LIN {X 0,Y 474.615,Z 281.367,A -85,B 0,C 180,E1 -7440.886,E2 -7440.886} C_VEL
LIN {X 0,Y 474.653,Z 281.359,A -85,B 0,C 180,E1 -7443.629,E2 -7443.629} C_VEL
LIN {X 0,Y 474.629,Z 281.364,A -85,B 0,C 180,E1 -7446.642,E2 -7446.642} C_VEL
LIN {X 0,Y 474.65,Z 281.358,A -85,B 0,C 180,E1 -7450.09,E2 -7450.09} C_VEL
LIN {X 0,Y 474.651,Z 281.358,A -85,B 0,C 180,E1 -7451.7,E2 -7451.7} C_VEL
LIN {X 0,Y 473.99,Z 281.443,A -85,B 0,C 180,E1 -7452.409,E2 -7452.409} C_VEL
LIN {X 0,Y 471.138,Z 281.798,A -85,B 0,C 180,E1 -7453.561,E2 -7453.561} C_VEL
LIN {X 0,Y 468.72,Z 282.101,A -85,B 0,C 180,E1 -7454.489,E2 -7454.489} C_VEL
LIN {X 0,Y 467.679,Z 282.229,A -85,B 0,C 180,E1 -7455.206,E2 -7455.206} C_VEL
LIN {X 0,Y 467.593,Z 282.238,A -85,B 0,C 180,E1 -7455.449,E2 -7455.449} C_VEL
LIN {X 0,Y 467.65,Z 282.234,A -85,B 0,C 180,E1 -7458.734,E2 -7458.734} C_VEL
LIN {X 0,Y 467.747,Z 282.218,A -85,B 0,C 180,E1 -7462.228,E2 -7462.228} C_VEL
LIN {X 0,Y 467.722,Z 282.226,A -85,B 0,C 180,E1 -7464.827,E2 -7464.827} C_VEL
LIN {X 0,Y 467.857,Z 282.206,A -85,B 0,C 180,E1 -7467.416,E2 -7467.416} C_VEL
LIN {X 0,Y 467.88,Z 282.201,A -85,B 0,C 180,E1 -7469.999,E2 -7469.999} C_VEL
LIN {X 0,Y 467.857,Z 282.206,A -85,B 0,C 180,E1 -7472.581,E2 -7472.581} C_VEL
LIN {X 0,Y 467.731,Z 282.219,A -85,B 0,C 180,E1 -7476.036,E2 -7476.036} C_VEL
LIN {X 0,Y 467.676,Z 282.228,A -85,B 0,C 180,E1 -7478.641,E2 -7478.641} C_VEL
LIN {X 0,Y 467.675,Z 282.226,A -85,B 0,C 180,E1 -7482.142,E2 -7482.142} C_VEL
LIN {X 0,Y 467.64,Z 282.231,A -85,B 0,C 180,E1 -7485.883,E2 -7485.883} C_VEL
LIN {X 0,Y 467.613,Z 282.238,A -85,B 0,C 180,E1 -7489.305,E2 -7489.305} C_VEL
LIN {X 0,Y 467.553,Z 282.241,A -85,B 0,C 180,E1 -7492.069,E2 -7492.069} C_VEL
LIN {X 0,Y 467.59,Z 282.241,A -85,B 0,C 180,E1 -7494.884,E2 -7494.884} C_VEL
LIN {X 0,Y 467.61,Z 282.235,A -85,B 0,C 180,E1 -7497.765,E2 -7497.765} C_VEL
LIN {X 0,Y 467.558,Z 282.246,A -85,B 0,C 180,E1 -7501.044,E2 -7501.044} C_VEL
LIN {X 0,Y 467.566,Z 282.239,A -85,B 0,C 180,E1 -7504.239,E2 -7504.239} C_VEL
LIN {X 0,Y 467.526,Z 282.252,A -85,B 0,C 180,E1 -7507.184,E2 -7507.184} C_VEL
LIN {X 0,Y 467.572,Z 282.24,A -85,B 0,C 180,E1 -7510.258,E2 -7510.258} C_VEL
LIN {X 0,Y 467.639,Z 282.299,A -85,B 0,C 180,E1 -7512.891,E2 -7512.891} C_VEL
LIN {X 0,Y 468.46,Z 287.03,A -85,B 0,C 180,E1 -7513.937,E2 -7513.937} C_VEL
LIN {X 0,Y 468.452,Z 292.664,A -85,B 0,C 180,E1 -7515.1,E2 -7515.1} C_VEL
LIN {X 0,Y 471.354,Z 307.156,A -85,B 0,C 180,E1 -7515.447,E2 -7515.447} C_VEL
LIN {X 0,Y 470.368,Z 400.533,A -85,B 0,C 180,E1 -7516.983,E2 -7516.983} C_VEL
LIN {X 0,Y 470.151,Z 413.603,A -85,B 0,C 180,E1 -7517.376,E2 -7517.376} C_VEL
LIN {X 0,Y 469.792,Z 425.843,A -85,B 0,C 180,E1 -7517.909,E2 -7517.909} C_VEL
LIN {X 0,Y 469.379,Z 437.833,A -85,B 0,C 180,E1 -7518.619,E2 -7518.619} C_VEL
LIN {X 0,Y 468.918,Z 448.857,A -85,B 0,C 180,E1 -7519.452,E2 -7519.452} C_VEL
LIN {X 0,Y 468.501,Z 458.862,A -85,B 0,C 180,E1 -7520.392,E2 -7520.392} C_VEL
LIN {X 0,Y 468.086,Z 468.527,A -85,B 0,C 180,E1 -7521.514,E2 -7521.514} C_VEL
LIN {X 0,Y 467.678,Z 477.339,A -85,B 0,C 180,E1 -7522.783,E2 -7522.783} C_VEL
LIN {X 0,Y 467.324,Z 484.669,A -85,B 0,C 180,E1 -7524.091,E2 -7524.091} C_VEL
LIN {X 0,Y 467.094,Z 490.987,A -85,B 0,C 180,E1 -7525.526,E2 -7525.526} C_VEL
LIN {X 0,Y 466.941,Z 495.005,A -85,B 0,C 180,E1 -7526.677,E2 -7526.677} C_VEL
LIN {X 0,Y 466.833,Z 498.969,A -85,B 0,C 180,E1 -7528.204,E2 -7528.204} C_VEL
LIN {X 0,Y 466.675,Z 500.847,A -85,B 0,C 180,E1 -7529.201,E2 -7529.201} C_VEL
LIN {X 0,Y 466.619,Z 502.698,A -85,B 0,C 180,E1 -7530.863,E2 -7530.863} C_VEL
LIN {X 0,Y 466.607,Z 503.037,A -85,B 0,C 180,E1 -7532.69,E2 -7532.69} C_VEL
LIN {X 0,Y 466.652,Z 502.053,A -85,B 0,C 180,E1 -7534.104,E2 -7534.104} C_VEL
LIN {X 0,Y 466.727,Z 500.735,A -85,B 0,C 180,E1 -7535.063,E2 -7535.063} C_VEL
LIN {X 0,Y 466.906,Z 497.465,A -85,B 0,C 180,E1 -7536.646,E2 -7536.646} C_VEL
LIN {X 0,Y 467.021,Z 493.781,A -85,B 0,C 180,E1 -7537.901,E2 -7537.901} C_VEL
LIN {X 0,Y 467.222,Z 488.421,A -85,B 0,C 180,E1 -7539.306,E2 -7539.306} C_VEL
LIN {X 0,Y 467.566,Z 481.593,A -85,B 0,C 180,E1 -7540.69,E2 -7540.69} C_VEL
LIN {X 0,Y 467.971,Z 473.014,A -85,B 0,C 180,E1 -7542.07,E2 -7542.07} C_VEL
LIN {X 0,Y 468.422,Z 464.162,A -85,B 0,C 180,E1 -7543.213,E2 -7543.213} C_VEL
LIN {X 0,Y 468.804,Z 454.996,A -85,B 0,C 180,E1 -7544.18,E2 -7544.18} C_VEL
LIN {X 0,Y 469.327,Z 443.665,A -85,B 0,C 180,E1 -7545.141,E2 -7545.141} C_VEL
LIN {X 0,Y 469.742,Z 431.9,A -85,B 0,C 180,E1 -7545.93,E2 -7545.93} C_VEL
LIN {X 0,Y 470.084,Z 419.99,A -85,B 0,C 180,E1 -7546.532,E2 -7546.532} C_VEL
LIN {X 0,Y 470.378,Z 407.324,A -85,B 0,C 180,E1 -7546.992,E2 -7546.992} C_VEL
LIN {X 0,Y 470.57,Z 395.176,A -85,B 0,C 180,E1 -7547.274,E2 -7547.274} C_VEL
LIN {X 0,Y 471.399,Z 305.966,A -85,B 0,C 180,E1 -7548.757,E2 -7548.757} C_VEL
LIN {X 0,Y 468.554,Z 292.044,A -85,B 0,C 180,E1 -7549.139,E2 -7549.139} C_VEL
LIN {X 0,Y 468.454,Z 286.338,A -85,B 0,C 180,E1 -7550.066,E2 -7550.066} C_VEL
LIN {X 0,Y 467.639,Z 282.237,A -85,B 0,C 180,E1 -7550.785,E2 -7550.785} C_VEL
LIN {X 0,Y 467.643,Z 282.237,A -85,B 0,C 180,E1 -7553.095,E2 -7553.095} C_VEL
LIN {X 0,Y 467.666,Z 282.236,A -85,B 0,C 180,E1 -7554.827,E2 -7554.827} C_VEL
LIN {X 0,Y 467.807,Z 282.215,A -85,B 0,C 180,E1 -7557.417,E2 -7557.417} C_VEL
LIN {X 0,Y 467.77,Z 282.221,A -85,B 0,C 180,E1 -7560.861,E2 -7560.861} C_VEL
LIN {X 0,Y 467.808,Z 282.214,A -85,B 0,C 180,E1 -7562.584,E2 -7562.584} C_VEL
LIN {X 0,Y 467.688,Z 282.225,A -85,B 0,C 180,E1 -7566.039,E2 -7566.039} C_VEL
LIN {X 0,Y 467.627,Z 282.235,A -85,B 0,C 180,E1 -7568.644,E2 -7568.644} C_VEL
LIN {X 0,Y 467.643,Z 282.23,A -85,B 0,C 180,E1 -7572.146,E2 -7572.146} C_VEL
LIN {X 0,Y 467.597,Z 282.235,A -85,B 0,C 180,E1 -7575.888,E2 -7575.888} C_VEL
LIN {X 0,Y 467.571,Z 282.241,A -85,B 0,C 180,E1 -7579.31,E2 -7579.31} C_VEL
LIN {X 0,Y 467.483,Z 282.249,A -85,B 0,C 180,E1 -7582.077,E2 -7582.077} C_VEL
LIN {X 0,Y 467.555,Z 282.246,A -85,B 0,C 180,E1 -7584.89,E2 -7584.89} C_VEL
LIN {X 0,Y 467.582,Z 282.238,A -85,B 0,C 180,E1 -7587.772,E2 -7587.772} C_VEL
LIN {X 0,Y 467.524,Z 282.25,A -85,B 0,C 180,E1 -7591.048,E2 -7591.048} C_VEL
LIN {X 0,Y 467.549,Z 282.239,A -85,B 0,C 180,E1 -7594.246,E2 -7594.246} C_VEL
LIN {X 0,Y 467.511,Z 282.25,A -85,B 0,C 180,E1 -7597.19,E2 -7597.19} C_VEL
LIN {X 0,Y 467.563,Z 282.239,A -85,B 0,C 180,E1 -7600.267,E2 -7600.267} C_VEL
LIN {X 0,Y 467.555,Z 282.239,A -85,B 0,C 180,E1 -7602.571,E2 -7602.571} C_VEL
LIN {X 0,Y 467.54,Z 282.246,A -85,B 0,C 180,E1 -7605.057,E2 -7605.057} C_VEL
LIN {X 0,Y 467.562,Z 282.246,A -85,B 0,C 180,E1 -7607.444,E2 -7607.444} C_VEL
LIN {X 0,Y 467.535,Z 282.246,A -85,B 0,C 180,E1 -7610.857,E2 -7610.857} C_VEL
LIN {X 0,Y 467.539,Z 282.246,A -85,B 0,C 180,E1 -7614.265,E2 -7614.265} C_VEL
LIN {X 0,Y 467.563,Z 282.251,A -85,B 0,C 180,E1 -7617.325,E2 -7617.325} C_VEL
LIN {X 0,Y 467.543,Z 282.248,A -85,B 0,C 180,E1 -7620.674,E2 -7620.674} C_VEL
LIN {X 0,Y 467.63,Z 282.33,A -85,B 0,C 180,E1 -7623.686,E2 -7623.686} C_VEL
LIN {X 0,Y 469.549,Z 292.668,A -85,B 0,C 180,E1 -7625.432,E2 -7625.432} C_VEL
LIN {X 0,Y 469.283,Z 306.157,A -85,B 0,C 180,E1 -7627.553,E2 -7627.553} C_VEL
LIN {X 0,Y 468.583,Z 327.553,A -85,B 0,C 180,E1 -7630.892,E2 -7630.892} C_VEL
LIN {X 0,Y 468.248,Z 340.575,A -85,B 0,C 180,E1 -7632.913,E2 -7632.913} C_VEL
LIN {X 0,Y 471.148,Z 362.036,A -85,B 0,C 180,E1 -7633.4,E2 -7633.4} C_VEL
LIN {X 0,Y 470.221,Z 450.57,A -85,B 0,C 180,E1 -7634.868,E2 -7634.868} C_VEL
LIN {X 0,Y 469.875,Z 464.289,A -85,B 0,C 180,E1 -7635.272,E2 -7635.272} C_VEL
LIN {X 0,Y 469.385,Z 476.739,A -85,B 0,C 180,E1 -7635.81,E2 -7635.81} C_VEL
LIN {X 0,Y 468.909,Z 489.513,A -85,B 0,C 180,E1 -7636.569,E2 -7636.569} C_VEL
LIN {X 0,Y 468.43,Z 501.178,A -85,B 0,C 180,E1 -7637.46,E2 -7637.46} C_VEL
LIN {X 0,Y 468.002,Z 511.192,A -85,B 0,C 180,E1 -7638.416,E2 -7638.416} C_VEL
LIN {X 0,Y 467.484,Z 521.296,A -85,B 0,C 180,E1 -7639.609,E2 -7639.609} C_VEL
LIN {X 0,Y 467.163,Z 530.213,A -85,B 0,C 180,E1 -7640.914,E2 -7640.914} C_VEL
LIN {X 0,Y 466.93,Z 537.327,A -85,B 0,C 180,E1 -7642.217,E2 -7642.217} C_VEL
LIN {X 0,Y 466.788,Z 543.23,A -85,B 0,C 180,E1 -7643.569,E2 -7643.569} C_VEL
LIN {X 0,Y 466.766,Z 547.525,A -85,B 0,C 180,E1 -7644.819,E2 -7644.819} C_VEL
LIN {X 0,Y 466.668,Z 549.898,A -85,B 0,C 180,E1 -7645.683,E2 -7645.683} C_VEL
LIN {X 0,Y 466.731,Z 551.835,A -85,B 0,C 180,E1 -7646.549,E2 -7646.549} C_VEL
LIN {X 0,Y 466.701,Z 553.285,A -85,B 0,C 180,E1 -7647.412,E2 -7647.412} C_VEL
LIN {X 0,Y 466.693,Z 554.326,A -85,B 0,C 180,E1 -7648.276,E2 -7648.276} C_VEL
LIN {X 0,Y 466.625,Z 554.964,A -85,B 0,C 180,E1 -7649.138,E2 -7649.138} C_VEL
LIN {X 0,Y 466.61,Z 555.198,A -85,B 0,C 180,E1 -7650.001,E2 -7650.001} C_VEL
LIN {X 0,Y 466.693,Z 554.379,A -85,B 0,C 180,E1 -7651.727,E2 -7651.727} C_VEL
LIN {X 0,Y 466.701,Z 553.37,A -85,B 0,C 180,E1 -7652.59,E2 -7652.59} C_VEL
LIN {X 0,Y 466.729,Z 551.936,A -85,B 0,C 180,E1 -7653.454,E2 -7653.454} C_VEL
LIN {X 0,Y 466.693,Z 548.933,A -85,B 0,C 180,E1 -7654.752,E2 -7654.752} C_VEL
LIN {X 0,Y 466.753,Z 544.861,A -85,B 0,C 180,E1 -7656.051,E2 -7656.051} C_VEL
LIN {X 0,Y 466.908,Z 538.583,A -85,B 0,C 180,E1 -7657.569,E2 -7657.569} C_VEL
LIN {X 0,Y 467.106,Z 531.735,A -85,B 0,C 180,E1 -7658.872,E2 -7658.872} C_VEL
LIN {X 0,Y 467.424,Z 523.218,A -85,B 0,C 180,E1 -7660.176,E2 -7660.176} C_VEL
LIN {X 0,Y 467.852,Z 514.443,A -85,B 0,C 180,E1 -7661.262,E2 -7661.262} C_VEL
LIN {X 0,Y 468.289,Z 504.35,A -85,B 0,C 180,E1 -7662.283,E2 -7662.283} C_VEL
LIN {X 0,Y 468.776,Z 492.901,A -85,B 0,C 180,E1 -7663.217,E2 -7663.217} C_VEL
LIN {X 0,Y 469.247,Z 480.88,A -85,B 0,C 180,E1 -7663.975,E2 -7663.975} C_VEL
LIN {X 0,Y 469.697,Z 468.412,A -85,B 0,C 180,E1 -7664.57,E2 -7664.57} C_VEL
LIN {X 0,Y 470.069,Z 455.524,A -85,B 0,C 180,E1 -7665.001,E2 -7665.001} C_VEL
LIN {X 0,Y 470.402,Z 440.405,A -85,B 0,C 180,E1 -7665.295,E2 -7665.295} C_VEL
LIN {X 0,Y 471.012,Z 361.47,A -85,B 0,C 180,E1 -7666.574,E2 -7666.574} C_VEL
LIN {X 0,Y 468.311,Z 342.083,A -85,B 0,C 180,E1 -7667.016,E2 -7667.016} C_VEL
LIN {X 0,Y 469.033,Z 322.86,A -85,B 0,C 180,E1 -7670.159,E2 -7670.159} C_VEL
LIN {X 0,Y 469.8,Z 304.956,A -85,B 0,C 180,E1 -7673.121,E2 -7673.121} C_VEL
LIN {X 0,Y 470.203,Z 295.306,A -85,B 0,C 180,E1 -7674.739,E2 -7674.739} C_VEL
LIN {X 0,Y 467.595,Z 282.241,A -85,B 0,C 180,E1 -7677.129,E2 -7677.129} C_VEL
LIN {X 0,Y 467.563,Z 282.247,A -85,B 0,C 180,E1 -7680.733,E2 -7680.733} C_VEL
LIN {X 0,Y 467.559,Z 282.24,A -85,B 0,C 180,E1 -7683.788,E2 -7683.788} C_VEL
LIN {X 0,Y 467.502,Z 282.251,A -85,B 0,C 180,E1 -7686.962,E2 -7686.962} C_VEL
LIN {X 0,Y 467.549,Z 282.242,A -85,B 0,C 180,E1 -7689.949,E2 -7689.949} C_VEL
LIN {X 0,Y 467.512,Z 282.251,A -85,B 0,C 180,E1 -7692.565,E2 -7692.565} C_VEL
LIN {X 0,Y 467.55,Z 282.244,A -85,B 0,C 180,E1 -7695.05,E2 -7695.05} C_VEL
LIN {X 0,Y 467.544,Z 282.249,A -85,B 0,C 180,E1 -7698.723,E2 -7698.723} C_VEL
LIN {X 0,Y 467.531,Z 282.244,A -85,B 0,C 180,E1 -7701.952,E2 -7701.952} C_VEL
LIN {X 0,Y 467.532,Z 282.246,A -85,B 0,C 180,E1 -7705.164,E2 -7705.164} C_VEL
LIN {X 0,Y 467.534,Z 282.246,A -85,B 0,C 180,E1 -7708.256,E2 -7708.256} C_VEL
LIN {X 0,Y 467.544,Z 282.244,A -85,B 0,C 180,E1 -7711.248,E2 -7711.248} C_VEL
LIN {X 0,Y 467.559,Z 282.243,A -85,B 0,C 180,E1 -7714.157,E2 -7714.157} C_VEL
LIN {X 0,Y 467.541,Z 282.248,A -85,B 0,C 180,E1 -7716.994,E2 -7716.994} C_VEL
LIN {X 0,Y 467.587,Z 282.237,A -85,B 0,C 180,E1 -7719.775,E2 -7719.775} C_VEL
LIN {X 0,Y 467.561,Z 282.243,A -85,B 0,C 180,E1 -7722.505,E2 -7722.505} C_VEL
LIN {X 0,Y 467.567,Z 282.243,A -85,B 0,C 180,E1 -7725.195,E2 -7725.195} C_VEL
LIN {X 0,Y 467.64,Z 282.231,A -85,B 0,C 180,E1 -7727.854,E2 -7727.854} C_VEL
LIN {X 0,Y 467.646,Z 282.232,A -85,B 0,C 180,E1 -7731.356,E2 -7731.356} C_VEL
LIN {X 0,Y 467.697,Z 282.225,A -85,B 0,C 180,E1 -7733.962,E2 -7733.962} C_VEL
LIN {X 0,Y 467.821,Z 282.21,A -85,B 0,C 180,E1 -7737.416,E2 -7737.416} C_VEL
LIN {X 0,Y 467.841,Z 282.207,A -85,B 0,C 180,E1 -7740,E2 -7740} C_VEL
LIN {X 0,Y 467.821,Z 282.211,A -85,B 0,C 180,E1 -7742.583,E2 -7742.583} C_VEL
LIN {X 0,Y 467.697,Z 282.225,A -85,B 0,C 180,E1 -7746.038,E2 -7746.038} C_VEL
LIN {X 0,Y 467.647,Z 282.233,A -85,B 0,C 180,E1 -7748.643,E2 -7748.643} C_VEL
LIN {X 0,Y 467.648,Z 282.231,A -85,B 0,C 180,E1 -7752.145,E2 -7752.145} C_VEL
LIN {X 0,Y 467.615,Z 282.235,A -85,B 0,C 180,E1 -7755.885,E2 -7755.885} C_VEL
LIN {X 0,Y 467.59,Z 282.241,A -85,B 0,C 180,E1 -7759.309,E2 -7759.309} C_VEL
LIN {X 0,Y 467.501,Z 282.249,A -85,B 0,C 180,E1 -7762.075,E2 -7762.075} C_VEL
LIN {X 0,Y 467.572,Z 282.243,A -85,B 0,C 180,E1 -7764.889,E2 -7764.889} C_VEL
LIN {X 0,Y 467.592,Z 282.238,A -85,B 0,C 180,E1 -7767.77,E2 -7767.77} C_VEL
LIN {X 0,Y 467.544,Z 282.247,A -85,B 0,C 180,E1 -7771.047,E2 -7771.047} C_VEL
LIN {X 0,Y 467.564,Z 282.242,A -85,B 0,C 180,E1 -7774.244,E2 -7774.244} C_VEL
LIN {X 0,Y 467.526,Z 282.249,A -85,B 0,C 180,E1 -7777.188,E2 -7777.188} C_VEL
LIN {X 0,Y 467.574,Z 282.241,A -85,B 0,C 180,E1 -7780.264,E2 -7780.264} C_VEL
LIN {X 0,Y 467.567,Z 282.244,A -85,B 0,C 180,E1 -7782.569,E2 -7782.569} C_VEL
LIN {X 0,Y 467.556,Z 282.243,A -85,B 0,C 180,E1 -7786.178,E2 -7786.178} C_VEL
LIN {X 0,Y 467.573,Z 282.244,A -85,B 0,C 180,E1 -7788.723,E2 -7788.723} C_VEL
LIN {X 0,Y 467.564,Z 282.244,A -85,B 0,C 180,E1 -7791.408,E2 -7791.408} C_VEL
LIN {X 0,Y 467.55,Z 282.244,A -85,B 0,C 180,E1 -7794.262,E2 -7794.262} C_VEL
LIN {X 0,Y 467.571,Z 282.243,A -85,B 0,C 180,E1 -7797.322,E2 -7797.322} C_VEL
LIN {X 0,Y 467.561,Z 282.245,A -85,B 0,C 180,E1 -7800.669,E2 -7800.669} C_VEL
LIN {X 0,Y 467.609,Z 282.238,A -85,B 0,C 180,E1 -7803.201,E2 -7803.201} C_VEL
LIN {X 0,Y 467.586,Z 282.24,A -85,B 0,C 180,E1 -7806.469,E2 -7806.469} C_VEL
LIN {X 0,Y 467.618,Z 282.235,A -85,B 0,C 180,E1 -7809.778,E2 -7809.778} C_VEL
LIN {X 0,Y 467.605,Z 282.238,A -85,B 0,C 180,E1 -7812.507,E2 -7812.507} C_VEL
LIN {X 0,Y 467.603,Z 282.239,A -85,B 0,C 180,E1 -7815.196,E2 -7815.196} C_VEL
LIN {X 0,Y 467.593,Z 282.238,A -85,B 0,C 180,E1 -7815.449,E2 -7815.449} C_VEL
LIN {X 0,Y 466.924,Z 282.321,A -85,B 0,C 180,E1 -7816.168,E2 -7816.168} C_VEL
LIN {X 0,Y 464.08,Z 282.677,A -85,B 0,C 180,E1 -7817.337,E2 -7817.337} C_VEL
LIN {X 0,Y 461.68,Z 282.974,A -85,B 0,C 180,E1 -7818.279,E2 -7818.279} C_VEL
LIN {X 0,Y 460.655,Z 283.105,A -85,B 0,C 180,E1 -7819.006,E2 -7819.006} C_VEL
LIN {X 0,Y 460.574,Z 283.112,A -85,B 0,C 180,E1 -7819.253,E2 -7819.253} C_VEL
LIN {X 0,Y 460.718,Z 283.095,A -85,B 0,C 180,E1 -7822.538,E2 -7822.538} C_VEL
LIN {X 0,Y 460.695,Z 283.1,A -85,B 0,C 180,E1 -7824.747,E2 -7824.747} C_VEL
LIN {X 0,Y 460.822,Z 283.082,A -85,B 0,C 180,E1 -7827.376,E2 -7827.376} C_VEL
LIN {X 0,Y 460.851,Z 283.077,A -85,B 0,C 180,E1 -7829.999,E2 -7829.999} C_VEL
LIN {X 0,Y 460.822,Z 283.083,A -85,B 0,C 180,E1 -7832.621,E2 -7832.621} C_VEL
LIN {X 0,Y 460.697,Z 283.096,A -85,B 0,C 180,E1 -7836.128,E2 -7836.128} C_VEL
LIN {X 0,Y 460.623,Z 283.108,A -85,B 0,C 180,E1 -7838.774,E2 -7838.774} C_VEL
LIN {X 0,Y 460.627,Z 283.105,A -85,B 0,C 180,E1 -7842.454,E2 -7842.454} C_VEL
LIN {X 0,Y 460.59,Z 283.109,A -85,B 0,C 180,E1 -7845.995,E2 -7845.995} C_VEL
LIN {X 0,Y 460.56,Z 283.117,A -85,B 0,C 180,E1 -7848.899,E2 -7848.899} C_VEL
LIN {X 0,Y 460.55,Z 283.116,A -85,B 0,C 180,E1 -7851.48,E2 -7851.48} C_VEL
LIN {X 0,Y 460.529,Z 283.116,A -85,B 0,C 180,E1 -7854.329,E2 -7854.329} C_VEL
LIN {X 0,Y 460.567,Z 283.117,A -85,B 0,C 180,E1 -7857.24,E2 -7857.24} C_VEL
LIN {X 0,Y 460.51,Z 283.118,A -85,B 0,C 180,E1 -7860.235,E2 -7860.235} C_VEL
LIN {X 0,Y 460.506,Z 283.124,A -85,B 0,C 180,E1 -7863.321,E2 -7863.321} C_VEL
LIN {X 0,Y 460.454,Z 283.125,A -85,B 0,C 180,E1 -7866.525,E2 -7866.525} C_VEL
LIN {X 0,Y 460.556,Z 283.116,A -85,B 0,C 180,E1 -7869.853,E2 -7869.853} C_VEL
LIN {X 0,Y 460.595,Z 283.191,A -85,B 0,C 180,E1 -7872.732,E2 -7872.732} C_VEL
LIN {X 0,Y 461.493,Z 289.015,A -85,B 0,C 180,E1 -7874.031,E2 -7874.031} C_VEL
LIN {X 0,Y 461.462,Z 292.957,A -85,B 0,C 180,E1 -7874.849,E2 -7874.849} C_VEL
LIN {X 0,Y 464.515,Z 307.983,A -85,B 0,C 180,E1 -7875.22,E2 -7875.22} C_VEL
LIN {X 0,Y 463.472,Z 400.889,A -85,B 0,C 180,E1 -7876.778,E2 -7876.778} C_VEL
LIN {X 0,Y 463.242,Z 413.709,A -85,B 0,C 180,E1 -7877.168,E2 -7877.168} C_VEL
LIN {X 0,Y 462.887,Z 426.171,A -85,B 0,C 180,E1 -7877.718,E2 -7877.718} C_VEL
LIN {X 0,Y 462.443,Z 438.672,A -85,B 0,C 180,E1 -7878.472,E2 -7878.472} C_VEL
LIN {X 0,Y 461.921,Z 450.36,A -85,B 0,C 180,E1 -7879.381,E2 -7879.381} C_VEL
LIN {X 0,Y 461.542,Z 459.279,A -85,B 0,C 180,E1 -7880.243,E2 -7880.243} C_VEL
LIN {X 0,Y 461.102,Z 468.523,A -85,B 0,C 180,E1 -7881.325,E2 -7881.325} C_VEL
LIN {X 0,Y 460.704,Z 476.586,A -85,B 0,C 180,E1 -7882.481,E2 -7882.481} C_VEL
LIN {X 0,Y 460.366,Z 483.958,A -85,B 0,C 180,E1 -7883.778,E2 -7883.778} C_VEL
LIN {X 0,Y 460.066,Z 490.893,A -85,B 0,C 180,E1 -7885.318,E2 -7885.318} C_VEL
LIN {X 0,Y 459.873,Z 495.416,A -85,B 0,C 180,E1 -7886.622,E2 -7886.622} C_VEL
LIN {X 0,Y 459.754,Z 499.378,A -85,B 0,C 180,E1 -7888.172,E2 -7888.172} C_VEL
LIN {X 0,Y 459.54,Z 501.956,A -85,B 0,C 180,E1 -7889.69,E2 -7889.69} C_VEL
LIN {X 0,Y 459.525,Z 503,A -85,B 0,C 180,E1 -7890.699,E2 -7890.699} C_VEL
LIN {X 0,Y 459.509,Z 503.458,A -85,B 0,C 180,E1 -7891.698,E2 -7891.698} C_VEL
LIN {X 0,Y 459.519,Z 503.443,A -85,B 0,C 180,E1 -7892.689,E2 -7892.689} C_VEL
LIN {X 0,Y 459.606,Z 502.104,A -85,B 0,C 180,E1 -7894.432,E2 -7894.432} C_VEL
LIN {X 0,Y 459.719,Z 500.287,A -85,B 0,C 180,E1 -7895.622,E2 -7895.622} C_VEL
LIN {X 0,Y 459.886,Z 496.984,A -85,B 0,C 180,E1 -7897.065,E2 -7897.065} C_VEL
LIN {X 0,Y 460.081,Z 491.721,A -85,B 0,C 180,E1 -7898.7,E2 -7898.7} C_VEL
LIN {X 0,Y 460.385,Z 485.528,A -85,B 0,C 180,E1 -7900.145,E2 -7900.145} C_VEL
LIN {X 0,Y 460.755,Z 477.822,A -85,B 0,C 180,E1 -7901.549,E2 -7901.549} C_VEL
LIN {X 0,Y 461.183,Z 469.913,A -85,B 0,C 180,E1 -7902.713,E2 -7902.713} C_VEL
LIN {X 0,Y 461.647,Z 460.602,A -85,B 0,C 180,E1 -7903.835,E2 -7903.835} C_VEL
LIN {X 0,Y 462.134,Z 450.778,A -85,B 0,C 180,E1 -7904.792,E2 -7904.792} C_VEL
LIN {X 0,Y 462.627,Z 439.041,A -85,B 0,C 180,E1 -7905.709,E2 -7905.709} C_VEL
LIN {X 0,Y 463.069,Z 427.286,A -85,B 0,C 180,E1 -7906.423,E2 -7906.423} C_VEL
LIN {X 0,Y 463.343,Z 413.994,A -85,B 0,C 180,E1 -7907.017,E2 -7907.017} C_VEL
LIN {X 0,Y 463.642,Z 400.585,A -85,B 0,C 180,E1 -7907.415,E2 -7907.415} C_VEL
LIN {X 0,Y 464.786,Z 307.882,A -85,B 0,C 180,E1 -7908.995,E2 -7908.995} C_VEL
LIN {X 0,Y 461.665,Z 292.463,A -85,B 0,C 180,E1 -7909.419,E2 -7909.419} C_VEL
LIN {X 0,Y 461.373,Z 286.866,A -85,B 0,C 180,E1 -7910.354,E2 -7910.354} C_VEL
LIN {X 0,Y 460.58,Z 283.116,A -85,B 0,C 180,E1 -7911.03,E2 -7911.03} C_VEL
LIN {X 0,Y 460.608,Z 283.113,A -85,B 0,C 180,E1 -7912.989,E2 -7912.989} C_VEL
LIN {X 0,Y 460.638,Z 283.111,A -85,B 0,C 180,E1 -7914.748,E2 -7914.748} C_VEL
LIN {X 0,Y 460.773,Z 283.092,A -85,B 0,C 180,E1 -7917.378,E2 -7917.378} C_VEL
LIN {X 0,Y 460.792,Z 283.084,A -85,B 0,C 180,E1 -7920,E2 -7920} C_VEL
LIN {X 0,Y 460.773,Z 283.091,A -85,B 0,C 180,E1 -7922.623,E2 -7922.623} C_VEL
LIN {X 0,Y 460.653,Z 283.101,A -85,B 0,C 180,E1 -7926.131,E2 -7926.131} C_VEL
LIN {X 0,Y 460.575,Z 283.114,A -85,B 0,C 180,E1 -7928.778,E2 -7928.778} C_VEL
LIN {X 0,Y 460.581,Z 283.111,A -85,B 0,C 180,E1 -7932.459,E2 -7932.459} C_VEL
LIN {X 0,Y 460.548,Z 283.113,A -85,B 0,C 180,E1 -7936,E2 -7936} C_VEL
LIN {X 0,Y 460.518,Z 283.121,A -85,B 0,C 180,E1 -7938.904,E2 -7938.904} C_VEL
LIN {X 0,Y 460.466,Z 283.126,A -85,B 0,C 180,E1 -7941.488,E2 -7941.488} C_VEL
LIN {X 0,Y 460.494,Z 283.12,A -85,B 0,C 180,E1 -7944.335,E2 -7944.335} C_VEL
LIN {X 0,Y 460.535,Z 283.122,A -85,B 0,C 180,E1 -7947.247,E2 -7947.247} C_VEL
LIN {X 0,Y 460.466,Z 283.124,A -85,B 0,C 180,E1 -7950.244,E2 -7950.244} C_VEL
LIN {X 0,Y 460.488,Z 283.125,A -85,B 0,C 180,E1 -7953.329,E2 -7953.329} C_VEL
LIN {X 0,Y 460.44,Z 283.128,A -85,B 0,C 180,E1 -7956.533,E2 -7956.533} C_VEL
LIN {X 0,Y 460.543,Z 283.115,A -85,B 0,C 180,E1 -7959.862,E2 -7959.862} C_VEL
LIN {X 0,Y 460.482,Z 283.123,A -85,B 0,C 180,E1 -7962.904,E2 -7962.904} C_VEL
LIN {X 0,Y 460.482,Z 283.124,A -85,B 0,C 180,E1 -7965.835,E2 -7965.835} C_VEL
LIN {X 0,Y 460.505,Z 283.123,A -85,B 0,C 180,E1 -7968.993,E2 -7968.993} C_VEL
LIN {X 0,Y 460.494,Z 283.127,A -85,B 0,C 180,E1 -7971.27,E2 -7971.27} C_VEL
LIN {X 0,Y 460.49,Z 283.124,A -85,B 0,C 180,E1 -7974.558,E2 -7974.558} C_VEL
LIN {X 0,Y 460.513,Z 283.128,A -85,B 0,C 180,E1 -7977.72,E2 -7977.72} C_VEL
LIN {X 0,Y 460.513,Z 283.125,A -85,B 0,C 180,E1 -7980.772,E2 -7980.772} C_VEL
LIN {X 0,Y 460.562,Z 283.215,A -85,B 0,C 180,E1 -7983.465,E2 -7983.465} C_VEL
LIN {X 0,Y 462.668,Z 294.216,A -85,B 0,C 180,E1 -7985.361,E2 -7985.361} C_VEL
LIN {X 0,Y 462.271,Z 308.685,A -85,B 0,C 180,E1 -7987.665,E2 -7987.665} C_VEL
LIN {X 0,Y 461.565,Z 329.991,A -85,B 0,C 180,E1 -7991.04,E2 -7991.04} C_VEL
LIN {X 0,Y 461.305,Z 340.355,A -85,B 0,C 180,E1 -7992.637,E2 -7992.637} C_VEL
LIN {X 0,Y 464.331,Z 362.558,A -85,B 0,C 180,E1 -7993.148,E2 -7993.148} C_VEL
LIN {X 0,Y 463.376,Z 450.164,A -85,B 0,C 180,E1 -7994.639,E2 -7994.639} C_VEL
LIN {X 0,Y 463.016,Z 463.857,A -85,B 0,C 180,E1 -7995.049,E2 -7995.049} C_VEL
LIN {X 0,Y 462.495,Z 476.302,A -85,B 0,C 180,E1 -7995.595,E2 -7995.595} C_VEL
LIN {X 0,Y 462.028,Z 487.48,A -85,B 0,C 180,E1 -7996.253,E2 -7996.253} C_VEL
LIN {X 0,Y 461.48,Z 499.455,A -85,B 0,C 180,E1 -7997.158,E2 -7997.158} C_VEL
LIN {X 0,Y 461.053,Z 509.726,A -85,B 0,C 180,E1 -7998.127,E2 -7998.127} C_VEL
LIN {X 0,Y 460.571,Z 519.221,A -85,B 0,C 180,E1 -7999.229,E2 -7999.229} C_VEL
LIN {X 0,Y 460.152,Z 528.424,A -85,B 0,C 180,E1 -8000.552,E2 -8000.552} C_VEL
LIN {X 0,Y 459.907,Z 535.855,A -85,B 0,C 180,E1 -8001.876,E2 -8001.876} C_VEL
LIN {X 0,Y 459.74,Z 540.874,A -85,B 0,C 180,E1 -8002.978,E2 -8002.978} C_VEL
LIN {X 0,Y 459.667,Z 545.759,A -85,B 0,C 180,E1 -8004.298,E2 -8004.298} C_VEL
LIN {X 0,Y 459.583,Z 549.498,A -85,B 0,C 180,E1 -8005.617,E2 -8005.617} C_VEL
LIN {X 0,Y 459.628,Z 551.435,A -85,B 0,C 180,E1 -8006.495,E2 -8006.495} C_VEL
LIN {X 0,Y 459.621,Z 552.889,A -85,B 0,C 180,E1 -8007.372,E2 -8007.372} C_VEL
LIN {X 0,Y 459.614,Z 553.93,A -85,B 0,C 180,E1 -8008.249,E2 -8008.249} C_VEL
LIN {X 0,Y 459.558,Z 554.57,A -85,B 0,C 180,E1 -8009.125,E2 -8009.125} C_VEL
LIN {X 0,Y 459.541,Z 554.802,A -85,B 0,C 180,E1 -8010.001,E2 -8010.001} C_VEL
LIN {X 0,Y 459.558,Z 554.59,A -85,B 0,C 180,E1 -8010.878,E2 -8010.878} C_VEL
LIN {X 0,Y 459.614,Z 553.981,A -85,B 0,C 180,E1 -8011.754,E2 -8011.754} C_VEL
LIN {X 0,Y 459.622,Z 552.969,A -85,B 0,C 180,E1 -8012.63,E2 -8012.63} C_VEL
LIN {X 0,Y 459.626,Z 551.529,A -85,B 0,C 180,E1 -8013.508,E2 -8013.508} C_VEL
LIN {X 0,Y 459.624,Z 548.518,A -85,B 0,C 180,E1 -8014.825,E2 -8014.825} C_VEL
LIN {X 0,Y 459.716,Z 543.365,A -85,B 0,C 180,E1 -8016.432,E2 -8016.432} C_VEL
LIN {X 0,Y 459.871,Z 537.106,A -85,B 0,C 180,E1 -8017.906,E2 -8017.906} C_VEL
LIN {X 0,Y 460.108,Z 529.974,A -85,B 0,C 180,E1 -8019.23,E2 -8019.23} C_VEL
LIN {X 0,Y 460.475,Z 521.047,A -85,B 0,C 180,E1 -8020.554,E2 -8020.554} C_VEL
LIN {X 0,Y 460.999,Z 510.903,A -85,B 0,C 180,E1 -8021.766,E2 -8021.766} C_VEL
LIN {X 0,Y 461.453,Z 500.643,A -85,B 0,C 180,E1 -8022.748,E2 -8022.748} C_VEL
LIN {X 0,Y 461.986,Z 489.02,A -85,B 0,C 180,E1 -8023.639,E2 -8023.639} C_VEL
LIN {X 0,Y 462.469,Z 477.05,A -85,B 0,C 180,E1 -8024.353,E2 -8024.353} C_VEL
LIN {X 0,Y 462.946,Z 463.827,A -85,B 0,C 180,E1 -8024.928,E2 -8024.928} C_VEL
LIN {X 0,Y 463.296,Z 450.822,A -85,B 0,C 180,E1 -8025.31,E2 -8025.31} C_VEL
LIN {X 0,Y 464.163,Z 362.041,A -85,B 0,C 180,E1 -8026.793,E2 -8026.793} C_VEL
LIN {X 0,Y 461.323,Z 341.751,A -85,B 0,C 180,E1 -8027.266,E2 -8027.266} C_VEL
LIN {X 0,Y 462.048,Z 323.805,A -85,B 0,C 180,E1 -8030.245,E2 -8030.245} C_VEL
LIN {X 0,Y 462.965,Z 304.553,A -85,B 0,C 180,E1 -8033.483,E2 -8033.483} C_VEL
LIN {X 0,Y 463.294,Z 297.202,A -85,B 0,C 180,E1 -8034.732,E2 -8034.732} C_VEL
LIN {X 0,Y 460.68,Z 283.635,A -85,B 0,C 180,E1 -8037.236,E2 -8037.236} C_VEL
LIN {X 0,Y 460.556,Z 283.116,A -85,B 0,C 180,E1 -8037.406,E2 -8037.406} C_VEL
LIN {X 0,Y 460.502,Z 283.124,A -85,B 0,C 180,E1 -8040.239,E2 -8040.239} C_VEL
LIN {X 0,Y 460.51,Z 283.118,A -85,B 0,C 180,E1 -8043.324,E2 -8043.324} C_VEL
LIN {X 0,Y 460.456,Z 283.13,A -85,B 0,C 180,E1 -8046.529,E2 -8046.529} C_VEL
LIN {X 0,Y 460.499,Z 283.12,A -85,B 0,C 180,E1 -8049.863,E2 -8049.863} C_VEL
LIN {X 0,Y 460.453,Z 283.13,A -85,B 0,C 180,E1 -8052.892,E2 -8052.892} C_VEL
LIN {X 0,Y 460.488,Z 283.121,A -85,B 0,C 180,E1 -8055.829,E2 -8055.829} C_VEL
LIN {X 0,Y 460.498,Z 283.124,A -85,B 0,C 180,E1 -8058.985,E2 -8058.985} C_VEL
LIN {X 0,Y 460.473,Z 283.126,A -85,B 0,C 180,E1 -8062.374,E2 -8062.374} C_VEL
LIN {X 0,Y 460.513,Z 283.118,A -85,B 0,C 180,E1 -8065.62,E2 -8065.62} C_VEL
LIN {X 0,Y 460.48,Z 283.128,A -85,B 0,C 180,E1 -8068.74,E2 -8068.74} C_VEL
LIN {X 0,Y 460.522,Z 283.117,A -85,B 0,C 180,E1 -8071.765,E2 -8071.765} C_VEL
LIN {X 0,Y 460.5,Z 283.125,A -85,B 0,C 180,E1 -8074.702,E2 -8074.702} C_VEL
LIN {X 0,Y 460.476,Z 283.124,A -85,B 0,C 180,E1 -8077.569,E2 -8077.569} C_VEL
LIN {X 0,Y 460.534,Z 283.118,A -85,B 0,C 180,E1 -8080.383,E2 -8080.383} C_VEL
LIN {X 0,Y 460.574,Z 283.112,A -85,B 0,C 180,E1 -8084.057,E2 -8084.057} C_VEL
LIN {X 0,Y 460.589,Z 283.11,A -85,B 0,C 180,E1 -8087.665,E2 -8087.665} C_VEL
LIN {X 0,Y 460.594,Z 283.112,A -85,B 0,C 180,E1 -8091.223,E2 -8091.223} C_VEL
LIN {X 0,Y 460.663,Z 283.101,A -85,B 0,C 180,E1 -8093.869,E2 -8093.869} C_VEL
LIN {X 0,Y 460.762,Z 283.09,A -85,B 0,C 180,E1 -8097.377,E2 -8097.377} C_VEL
LIN {X 0,Y 460.812,Z 283.082,A -85,B 0,C 180,E1 -8100,E2 -8100} C_VEL
LIN {X 0,Y 460.762,Z 283.091,A -85,B 0,C 180,E1 -8102.622,E2 -8102.622} C_VEL
LIN {X 0,Y 460.663,Z 283.102,A -85,B 0,C 180,E1 -8106.13,E2 -8106.13} C_VEL
LIN {X 0,Y 460.595,Z 283.112,A -85,B 0,C 180,E1 -8108.776,E2 -8108.776} C_VEL
LIN {X 0,Y 460.601,Z 283.111,A -85,B 0,C 180,E1 -8112.457,E2 -8112.457} C_VEL
LIN {X 0,Y 460.568,Z 283.113,A -85,B 0,C 180,E1 -8115.998,E2 -8115.998} C_VEL
LIN {X 0,Y 460.537,Z 283.119,A -85,B 0,C 180,E1 -8118.902,E2 -8118.902} C_VEL
LIN {X 0,Y 460.484,Z 283.125,A -85,B 0,C 180,E1 -8121.487,E2 -8121.487} C_VEL
LIN {X 0,Y 460.511,Z 283.122,A -85,B 0,C 180,E1 -8124.333,E2 -8124.333} C_VEL
LIN {X 0,Y 460.544,Z 283.12,A -85,B 0,C 180,E1 -8127.245,E2 -8127.245} C_VEL
LIN {X 0,Y 460.498,Z 283.123,A -85,B 0,C 180,E1 -8130.24,E2 -8130.24} C_VEL
LIN {X 0,Y 460.503,Z 283.124,A -85,B 0,C 180,E1 -8133.326,E2 -8133.326} C_VEL
LIN {X 0,Y 460.454,Z 283.13,A -85,B 0,C 180,E1 -8136.531,E2 -8136.531} C_VEL
LIN {X 0,Y 460.555,Z 283.115,A -85,B 0,C 180,E1 -8139.859,E2 -8139.859} C_VEL
LIN {X 0,Y 460.493,Z 283.125,A -85,B 0,C 180,E1 -8142.902,E2 -8142.902} C_VEL
LIN {X 0,Y 460.505,Z 283.121,A -85,B 0,C 180,E1 -8145.83,E2 -8145.83} C_VEL
LIN {X 0,Y 460.527,Z 283.12,A -85,B 0,C 180,E1 -8148.992,E2 -8148.992} C_VEL
LIN {X 0,Y 460.533,Z 283.12,A -85,B 0,C 180,E1 -8151.27,E2 -8151.27} C_VEL
LIN {X 0,Y 460.501,Z 283.124,A -85,B 0,C 180,E1 -8154.556,E2 -8154.556} C_VEL
LIN {X 0,Y 460.52,Z 283.119,A -85,B 0,C 180,E1 -8157.717,E2 -8157.717} C_VEL
LIN {X 0,Y 460.531,Z 283.122,A -85,B 0,C 180,E1 -8160.77,E2 -8160.77} C_VEL
LIN {X 0,Y 460.556,Z 283.115,A -85,B 0,C 180,E1 -8163.736,E2 -8163.736} C_VEL
LIN {X 0,Y 460.54,Z 283.119,A -85,B 0,C 180,E1 -8166.625,E2 -8166.625} C_VEL
LIN {X 0,Y 460.546,Z 283.117,A -85,B 0,C 180,E1 -8169.453,E2 -8169.453} C_VEL
LIN {X 0,Y 460.555,Z 283.114,A -85,B 0,C 180,E1 -8172.23,E2 -8172.23} C_VEL
LIN {X 0,Y 460.562,Z 283.117,A -85,B 0,C 180,E1 -8174.965,E2 -8174.965} C_VEL
LIN {X 0,Y 460.608,Z 283.109,A -85,B 0,C 180,E1 -8178.559,E2 -8178.559} C_VEL
LIN {X 0,Y 460.574,Z 283.112,A -85,B 0,C 180,E1 -8179.253,E2 -8179.253} C_VEL
LIN {X 0,Y 459.921,Z 283.197,A -85,B 0,C 180,E1 -8179.983,E2 -8179.983} C_VEL
LIN {X 0,Y 457.103,Z 283.553,A -85,B 0,C 180,E1 -8181.17,E2 -8181.17} C_VEL
LIN {X 0,Y 454.723,Z 283.849,A -85,B 0,C 180,E1 -8182.127,E2 -8182.127} C_VEL
LIN {X 0,Y 453.712,Z 283.972,A -85,B 0,C 180,E1 -8182.866,E2 -8182.866} C_VEL
LIN {X 0,Y 453.635,Z 283.979,A -85,B 0,C 180,E1 -8183.116,E2 -8183.116} C_VEL
LIN {X 0,Y 453.669,Z 283.975,A -85,B 0,C 180,E1 -8184.666,E2 -8184.666} C_VEL
LIN {X 0,Y 453.762,Z 283.962,A -85,B 0,C 180,E1 -8187.336,E2 -8187.336} C_VEL
LIN {X 0,Y 453.821,Z 283.953,A -85,B 0,C 180,E1 -8189.999,E2 -8189.999} C_VEL
LIN {X 0,Y 453.762,Z 283.962,A -85,B 0,C 180,E1 -8192.662,E2 -8192.662} C_VEL
LIN {X 0,Y 453.665,Z 283.972,A -85,B 0,C 180,E1 -8196.223,E2 -8196.223} C_VEL
LIN {X 0,Y 453.587,Z 283.987,A -85,B 0,C 180,E1 -8198.911,E2 -8198.911} C_VEL
LIN {X 0,Y 453.594,Z 283.982,A -85,B 0,C 180,E1 -8202.548,E2 -8202.548} C_VEL
LIN {X 0,Y 453.535,Z 283.987,A -85,B 0,C 180,E1 -8206.193,E2 -8206.193} C_VEL
LIN {X 0,Y 453.51,Z 283.997,A -85,B 0,C 180,E1 -8209.038,E2 -8209.038} C_VEL
LIN {X 0,Y 453.488,Z 283.994,A -85,B 0,C 180,E1 -8211.832,E2 -8211.832} C_VEL
LIN {X 0,Y 453.5,Z 283.994,A -85,B 0,C 180,E1 -8214.731,E2 -8214.731} C_VEL
LIN {X 0,Y 453.52,Z 283.989,A -85,B 0,C 180,E1 -8217.958,E2 -8217.958} C_VEL
LIN {X 0,Y 453.464,Z 283.998,A -85,B 0,C 180,E1 -8220.755,E2 -8220.755} C_VEL
LIN {X 0,Y 453.454,Z 283.997,A -85,B 0,C 180,E1 -8223.909,E2 -8223.909} C_VEL
LIN {X 0,Y 453.446,Z 284.006,A -85,B 0,C 180,E1 -8227.184,E2 -8227.184} C_VEL
LIN {X 0,Y 453.508,Z 283.996,A -85,B 0,C 180,E1 -8229.441,E2 -8229.441} C_VEL
LIN {X 0,Y 453.568,Z 284.118,A -85,B 0,C 180,E1 -8232.587,E2 -8232.587} C_VEL
LIN {X 0,Y 454.527,Z 289.754,A -85,B 0,C 180,E1 -8233.855,E2 -8233.855} C_VEL
LIN {X 0,Y 454.511,Z 293.225,A -85,B 0,C 180,E1 -8234.595,E2 -8234.595} C_VEL
LIN {X 0,Y 457.678,Z 308.876,A -85,B 0,C 180,E1 -8234.989,E2 -8234.989} C_VEL
LIN {X 0,Y 456.598,Z 400.983,A -85,B 0,C 180,E1 -8236.561,E2 -8236.561} C_VEL
LIN {X 0,Y 456.343,Z 414.15,A -85,B 0,C 180,E1 -8236.966,E2 -8236.966} C_VEL
LIN {X 0,Y 455.942,Z 427.283,A -85,B 0,C 180,E1 -8237.561,E2 -8237.561} C_VEL
LIN {X 0,Y 455.518,Z 439.281,A -85,B 0,C 180,E1 -8238.305,E2 -8238.305} C_VEL
LIN {X 0,Y 454.993,Z 450.386,A -85,B 0,C 180,E1 -8239.18,E2 -8239.18} C_VEL
LIN {X 0,Y 454.508,Z 460.947,A -85,B 0,C 180,E1 -8240.225,E2 -8240.225} C_VEL
LIN {X 0,Y 453.986,Z 470.921,A -85,B 0,C 180,E1 -8241.458,E2 -8241.458} C_VEL
LIN {X 0,Y 453.637,Z 477.807,A -85,B 0,C 180,E1 -8242.493,E2 -8242.493} C_VEL
LIN {X 0,Y 453.256,Z 485.494,A -85,B 0,C 180,E1 -8243.899,E2 -8243.899} C_VEL
LIN {X 0,Y 453.001,Z 491.523,A -85,B 0,C 180,E1 -8245.301,E2 -8245.301} C_VEL
LIN {X 0,Y 452.791,Z 496.868,A -85,B 0,C 180,E1 -8246.935,E2 -8246.935} C_VEL
LIN {X 0,Y 452.675,Z 499.788,A -85,B 0,C 180,E1 -8248.139,E2 -8248.139} C_VEL
LIN {X 0,Y 452.514,Z 501.67,A -85,B 0,C 180,E1 -8249.168,E2 -8249.168} C_VEL
LIN {X 0,Y 452.461,Z 503.16,A -85,B 0,C 180,E1 -8250.427,E2 -8250.427} C_VEL
LIN {X 0,Y 452.415,Z 503.698,A -85,B 0,C 180,E1 -8251.213,E2 -8251.213} C_VEL
LIN {X 0,Y 452.435,Z 503.904,A -85,B 0,C 180,E1 -8252.289,E2 -8252.289} C_VEL
LIN {X 0,Y 452.457,Z 503.606,A -85,B 0,C 180,E1 -8253.228,E2 -8253.228} C_VEL
LIN {X 0,Y 452.504,Z 502.792,A -85,B 0,C 180,E1 -8254.251,E2 -8254.251} C_VEL
LIN {X 0,Y 452.571,Z 501.492,A -85,B 0,C 180,E1 -8255.211,E2 -8255.211} C_VEL
LIN {X 0,Y 452.781,Z 498.431,A -85,B 0,C 180,E1 -8256.742,E2 -8256.742} C_VEL
LIN {X 0,Y 452.928,Z 494.476,A -85,B 0,C 180,E1 -8258.137,E2 -8258.137} C_VEL
LIN {X 0,Y 453.175,Z 489.096,A -85,B 0,C 180,E1 -8259.578,E2 -8259.578} C_VEL
LIN {X 0,Y 453.572,Z 482.179,A -85,B 0,C 180,E1 -8261.011,E2 -8261.011} C_VEL
LIN {X 0,Y 454.031,Z 473.562,A -85,B 0,C 180,E1 -8262.432,E2 -8262.432} C_VEL
LIN {X 0,Y 454.55,Z 464.771,A -85,B 0,C 180,E1 -8263.594,E2 -8263.594} C_VEL
LIN {X 0,Y 455.033,Z 454.792,A -85,B 0,C 180,E1 -8264.663,E2 -8264.663} C_VEL
LIN {X 0,Y 455.604,Z 443.96,A -85,B 0,C 180,E1 -8265.598,E2 -8265.598} C_VEL
LIN {X 0,Y 456.018,Z 433.422,A -85,B 0,C 180,E1 -8266.325,E2 -8266.325} C_VEL
LIN {X 0,Y 456.407,Z 420.921,A -85,B 0,C 180,E1 -8266.986,E2 -8266.986} C_VEL
LIN {X 0,Y 456.733,Z 408.723,A -85,B 0,C 180,E1 -8267.447,E2 -8267.447} C_VEL
LIN {X 0,Y 456.955,Z 395.713,A -85,B 0,C 180,E1 -8267.763,E2 -8267.763} C_VEL
LIN {X 0,Y 457.963,Z 308.053,A -85,B 0,C 180,E1 -8269.281,E2 -8269.281} C_VEL
LIN {X 0,Y 454.812,Z 292.971,A -85,B 0,C 180,E1 -8269.708,E2 -8269.708} C_VEL
LIN {X 0,Y 454.563,Z 288.692,A -85,B 0,C 180,E1 -8270.433,E2 -8270.433} C_VEL
LIN {X 0,Y 453.554,Z 283.99,A -85,B 0,C 180,E1 -8271.255,E2 -8271.255} C_VEL
LIN {X 0,Y 453.613,Z 283.983,A -85,B 0,C 180,E1 -8273.774,E2 -8273.774} C_VEL
LIN {X 0,Y 453.714,Z 283.972,A -85,B 0,C 180,E1 -8277.337,E2 -8277.337} C_VEL
LIN {X 0,Y 453.763,Z 283.96,A -85,B 0,C 180,E1 -8280,E2 -8280} C_VEL
LIN {X 0,Y 453.714,Z 283.97,A -85,B 0,C 180,E1 -8282.664,E2 -8282.664} C_VEL
LIN {X 0,Y 453.621,Z 283.978,A -85,B 0,C 180,E1 -8286.227,E2 -8286.227} C_VEL
LIN {X 0,Y 453.539,Z 283.992,A -85,B 0,C 180,E1 -8288.915,E2 -8288.915} C_VEL
LIN {X 0,Y 453.549,Z 283.988,A -85,B 0,C 180,E1 -8292.553,E2 -8292.553} C_VEL
LIN {X 0,Y 453.493,Z 283.992,A -85,B 0,C 180,E1 -8296.198,E2 -8296.198} C_VEL
LIN {X 0,Y 453.468,Z 284.002,A -85,B 0,C 180,E1 -8299.042,E2 -8299.042} C_VEL
LIN {X 0,Y 453.427,Z 284.001,A -85,B 0,C 180,E1 -8301.839,E2 -8301.839} C_VEL
LIN {X 0,Y 453.466,Z 283.999,A -85,B 0,C 180,E1 -8304.738,E2 -8304.738} C_VEL
LIN {X 0,Y 453.492,Z 283.992,A -85,B 0,C 180,E1 -8307.964,E2 -8307.964} C_VEL
LIN {X 0,Y 453.423,Z 284.002,A -85,B 0,C 180,E1 -8311.528,E2 -8311.528} C_VEL
LIN {X 0,Y 453.449,Z 283.998,A -85,B 0,C 180,E1 -8314.781,E2 -8314.781} C_VEL
LIN {X 0,Y 453.448,Z 283.998,A -85,B 0,C 180,E1 -8318.314,E2 -8318.314} C_VEL
LIN {X 0,Y 453.484,Z 283.994,A -85,B 0,C 180,E1 -8320.611,E2 -8320.611} C_VEL
LIN {X 0,Y 453.435,Z 283.999,A -85,B 0,C 180,E1 -8324.225,E2 -8324.225} C_VEL
LIN {X 0,Y 453.436,Z 284.003,A -85,B 0,C 180,E1 -8327.009,E2 -8327.009} C_VEL
LIN {X 0,Y 453.469,Z 284.002,A -85,B 0,C 180,E1 -8329.413,E2 -8329.413} C_VEL
LIN {X 0,Y 453.43,Z 284.003,A -85,B 0,C 180,E1 -8332.814,E2 -8332.814} C_VEL
LIN {X 0,Y 453.457,Z 284.003,A -85,B 0,C 180,E1 -8336.091,E2 -8336.091} C_VEL
LIN {X 0,Y 453.46,Z 284.008,A -85,B 0,C 180,E1 -8339.244,E2 -8339.244} C_VEL
LIN {X 0,Y 453.495,Z 283.997,A -85,B 0,C 180,E1 -8342.299,E2 -8342.299} C_VEL
LIN {X 0,Y 453.518,Z 284.116,A -85,B 0,C 180,E1 -8343.237,E2 -8343.237} C_VEL
LIN {X 0,Y 455.696,Z 295.015,A -85,B 0,C 180,E1 -8345.153,E2 -8345.153} C_VEL
LIN {X 0,Y 455.508,Z 306.851,A -85,B 0,C 180,E1 -8347.076,E2 -8347.076} C_VEL
LIN {X 0,Y 454.659,Z 327.625,A -85,B 0,C 180,E1 -8350.411,E2 -8350.411} C_VEL
LIN {X 0,Y 454.34,Z 339.745,A -85,B 0,C 180,E1 -8352.332,E2 -8352.332} C_VEL
LIN {X 0,Y 457.606,Z 363.951,A -85,B 0,C 180,E1 -8352.905,E2 -8352.905} C_VEL
LIN {X 0,Y 456.543,Z 450.146,A -85,B 0,C 180,E1 -8354.404,E2 -8354.404} C_VEL
LIN {X 0,Y 456.131,Z 463.645,A -85,B 0,C 180,E1 -8354.818,E2 -8354.818} C_VEL
LIN {X 0,Y 455.608,Z 475.986,A -85,B 0,C 180,E1 -8355.372,E2 -8355.372} C_VEL
LIN {X 0,Y 455.037,Z 488.702,A -85,B 0,C 180,E1 -8356.152,E2 -8356.152} C_VEL
LIN {X 0,Y 454.49,Z 499.836,A -85,B 0,C 180,E1 -8357.025,E2 -8357.025} C_VEL
LIN {X 0,Y 454.018,Z 510.347,A -85,B 0,C 180,E1 -8358.054,E2 -8358.054} C_VEL
LIN {X 0,Y 453.455,Z 520.471,A -85,B 0,C 180,E1 -8359.284,E2 -8359.284} C_VEL
LIN {X 0,Y 453.035,Z 529.399,A -85,B 0,C 180,E1 -8360.628,E2 -8360.628} C_VEL
LIN {X 0,Y 452.816,Z 536.525,A -85,B 0,C 180,E1 -8361.973,E2 -8361.973} C_VEL
LIN {X 0,Y 452.636,Z 542.405,A -85,B 0,C 180,E1 -8363.36,E2 -8363.36} C_VEL
LIN {X 0,Y 452.585,Z 546.731,A -85,B 0,C 180,E1 -8364.656,E2 -8364.656} C_VEL
LIN {X 0,Y 452.503,Z 549.109,A -85,B 0,C 180,E1 -8365.548,E2 -8365.548} C_VEL
LIN {X 0,Y 452.526,Z 551.044,A -85,B 0,C 180,E1 -8366.44,E2 -8366.44} C_VEL
LIN {X 0,Y 452.544,Z 552.497,A -85,B 0,C 180,E1 -8367.331,E2 -8367.331} C_VEL
LIN {X 0,Y 452.523,Z 553.537,A -85,B 0,C 180,E1 -8368.222,E2 -8368.222} C_VEL
LIN {X 0,Y 452.493,Z 554.178,A -85,B 0,C 180,E1 -8369.112,E2 -8369.112} C_VEL
LIN {X 0,Y 452.474,Z 554.404,A -85,B 0,C 180,E1 -8370.001,E2 -8370.001} C_VEL
LIN {X 0,Y 452.493,Z 554.187,A -85,B 0,C 180,E1 -8370.891,E2 -8370.891} C_VEL
LIN {X 0,Y 452.524,Z 553.571,A -85,B 0,C 180,E1 -8371.781,E2 -8371.781} C_VEL
LIN {X 0,Y 452.544,Z 552.555,A -85,B 0,C 180,E1 -8372.672,E2 -8372.672} C_VEL
LIN {X 0,Y 452.526,Z 551.099,A -85,B 0,C 180,E1 -8373.563,E2 -8373.563} C_VEL
LIN {X 0,Y 452.555,Z 548.076,A -85,B 0,C 180,E1 -8374.901,E2 -8374.901} C_VEL
LIN {X 0,Y 452.612,Z 543.398,A -85,B 0,C 180,E1 -8376.397,E2 -8376.397} C_VEL
LIN {X 0,Y 452.76,Z 537.642,A -85,B 0,C 180,E1 -8377.807,E2 -8377.807} C_VEL
LIN {X 0,Y 453.013,Z 530.743,A -85,B 0,C 180,E1 -8379.15,E2 -8379.15} C_VEL
LIN {X 0,Y 453.354,Z 522.133,A -85,B 0,C 180,E1 -8380.495,E2 -8380.495} C_VEL
LIN {X 0,Y 453.84,Z 513.277,A -85,B 0,C 180,E1 -8381.614,E2 -8381.614} C_VEL
LIN {X 0,Y 454.364,Z 502.933,A -85,B 0,C 180,E1 -8382.68,E2 -8382.68} C_VEL
LIN {X 0,Y 454.803,Z 492.956,A -85,B 0,C 180,E1 -8383.516,E2 -8383.516} C_VEL
LIN {X 0,Y 455.334,Z 481.221,A -85,B 0,C 180,E1 -8384.297,E2 -8384.297} C_VEL
LIN {X 0,Y 455.854,Z 467.783,A -85,B 0,C 180,E1 -8384.965,E2 -8384.965} C_VEL
LIN {X 0,Y 456.294,Z 455.01,A -85,B 0,C 180,E1 -8385.408,E2 -8385.408} C_VEL
LIN {X 0,Y 456.617,Z 440.086,A -85,B 0,C 180,E1 -8385.711,E2 -8385.711} C_VEL
LIN {X 0,Y 457.31,Z 362.757,A -85,B 0,C 180,E1 -8387.015,E2 -8387.015} C_VEL
LIN {X 0,Y 454.324,Z 341.486,A -85,B 0,C 180,E1 -8387.51,E2 -8387.51} C_VEL
LIN {X 0,Y 455.063,Z 324.754,A -85,B 0,C 180,E1 -8390.333,E2 -8390.333} C_VEL
LIN {X 0,Y 456.026,Z 305.485,A -85,B 0,C 180,E1 -8393.621,E2 -8393.621} C_VEL
LIN {X 0,Y 456.361,Z 298.591,A -85,B 0,C 180,E1 -8394.811,E2 -8394.811} C_VEL
LIN {X 0,Y 453.626,Z 284.556,A -85,B 0,C 180,E1 -8397.445,E2 -8397.445} C_VEL
LIN {X 0,Y 453.5,Z 283.995,A -85,B 0,C 180,E1 -8397.578,E2 -8397.578} C_VEL
LIN {X 0,Y 453.462,Z 284.003,A -85,B 0,C 180,E1 -8400.759,E2 -8400.759} C_VEL
LIN {X 0,Y 453.459,Z 283.997,A -85,B 0,C 180,E1 -8403.912,E2 -8403.912} C_VEL
LIN {X 0,Y 453.43,Z 284.001,A -85,B 0,C 180,E1 -8407.189,E2 -8407.189} C_VEL
LIN {X 0,Y 453.459,Z 284.002,A -85,B 0,C 180,E1 -8410.61,E2 -8410.61} C_VEL
LIN {X 0,Y 453.444,Z 284,A -85,B 0,C 180,E1 -8414.22,E2 -8414.22} C_VEL
LIN {X 0,Y 453.41,Z 284.007,A -85,B 0,C 180,E1 -8416.998,E2 -8416.998} C_VEL
LIN {X 0,Y 453.453,Z 283.998,A -85,B 0,C 180,E1 -8419.411,E2 -8419.411} C_VEL
LIN {X 0,Y 453.426,Z 284.008,A -85,B 0,C 180,E1 -8422.807,E2 -8422.807} C_VEL
LIN {X 0,Y 453.443,Z 284,A -85,B 0,C 180,E1 -8426.084,E2 -8426.084} C_VEL
LIN {X 0,Y 453.435,Z 284.002,A -85,B 0,C 180,E1 -8429.237,E2 -8429.237} C_VEL
LIN {X 0,Y 453.506,Z 283.993,A -85,B 0,C 180,E1 -8432.295,E2 -8432.295} C_VEL
LIN {X 0,Y 453.462,Z 283.999,A -85,B 0,C 180,E1 -8435.262,E2 -8435.262} C_VEL
LIN {X 0,Y 453.451,Z 284,A -85,B 0,C 180,E1 -8438.414,E2 -8438.414} C_VEL
LIN {X 0,Y 453.493,Z 283.998,A -85,B 0,C 180,E1 -8441.007,E2 -8441.007} C_VEL
LIN {X 0,Y 453.539,Z 283.988,A -85,B 0,C 180,E1 -8443.878,E2 -8443.878} C_VEL
LIN {X 0,Y 453.532,Z 283.99,A -85,B 0,C 180,E1 -8447.47,E2 -8447.47} C_VEL
LIN {X 0,Y 453.558,Z 283.99,A -85,B 0,C 180,E1 -8451.086,E2 -8451.086} C_VEL
LIN {X 0,Y 453.631,Z 283.977,A -85,B 0,C 180,E1 -8453.774,E2 -8453.774} C_VEL
LIN {X 0,Y 453.707,Z 283.969,A -85,B 0,C 180,E1 -8457.336,E2 -8457.336} C_VEL
LIN {X 0,Y 453.783,Z 283.958,A -85,B 0,C 180,E1 -8460,E2 -8460} C_VEL
LIN {X 0,Y 453.707,Z 283.969,A -85,B 0,C 180,E1 -8462.663,E2 -8462.663} C_VEL
LIN {X 0,Y 453.631,Z 283.978,A -85,B 0,C 180,E1 -8466.225,E2 -8466.225} C_VEL
LIN {X 0,Y 453.559,Z 283.989,A -85,B 0,C 180,E1 -8468.914,E2 -8468.914} C_VEL
LIN {X 0,Y 453.569,Z 283.987,A -85,B 0,C 180,E1 -8472.551,E2 -8472.551} C_VEL
LIN {X 0,Y 453.513,Z 283.993,A -85,B 0,C 180,E1 -8476.197,E2 -8476.197} C_VEL
LIN {X 0,Y 453.487,Z 283.998,A -85,B 0,C 180,E1 -8479.04,E2 -8479.04} C_VEL
LIN {X 0,Y 453.445,Z 284,A -85,B 0,C 180,E1 -8481.837,E2 -8481.837} C_VEL
LIN {X 0,Y 453.483,Z 283.997,A -85,B 0,C 180,E1 -8484.736,E2 -8484.736} C_VEL
LIN {X 0,Y 453.505,Z 283.993,A -85,B 0,C 180,E1 -8487.961,E2 -8487.961} C_VEL
LIN {X 0,Y 453.456,Z 284.001,A -85,B 0,C 180,E1 -8490.76,E2 -8490.76} C_VEL
LIN {X 0,Y 453.452,Z 284,A -85,B 0,C 180,E1 -8493.914,E2 -8493.914} C_VEL
LIN {X 0,Y 453.447,Z 284.002,A -85,B 0,C 180,E1 -8497.19,E2 -8497.19} C_VEL
LIN {X 0,Y 453.51,Z 283.994,A -85,B 0,C 180,E1 -8499.447,E2 -8499.447} C_VEL
LIN {X 0,Y 453.443,Z 284.002,A -85,B 0,C 180,E1 -8502.997,E2 -8502.997} C_VEL
LIN {X 0,Y 453.459,Z 283.999,A -85,B 0,C 180,E1 -8505.782,E2 -8505.782} C_VEL
LIN {X 0,Y 453.48,Z 283.997,A -85,B 0,C 180,E1 -8508.213,E2 -8508.213} C_VEL
LIN {X 0,Y 453.518,Z 283.994,A -85,B 0,C 180,E1 -8510.789,E2 -8510.789} C_VEL
LIN {X 0,Y 453.445,Z 284,A -85,B 0,C 180,E1 -8513.919,E2 -8513.919} C_VEL
LIN {X 0,Y 453.472,Z 283.999,A -85,B 0,C 180,E1 -8517.152,E2 -8517.152} C_VEL
LIN {X 0,Y 453.465,Z 283.998,A -85,B 0,C 180,E1 -8520.269,E2 -8520.269} C_VEL
LIN {X 0,Y 453.499,Z 283.995,A -85,B 0,C 180,E1 -8523.295,E2 -8523.295} C_VEL
LIN {X 0,Y 453.496,Z 283.994,A -85,B 0,C 180,E1 -8526.239,E2 -8526.239} C_VEL
LIN {X 0,Y 453.477,Z 283.998,A -85,B 0,C 180,E1 -8529.118,E2 -8529.118} C_VEL
LIN {X 0,Y 453.507,Z 283.992,A -85,B 0,C 180,E1 -8531.945,E2 -8531.945} C_VEL
LIN {X 0,Y 453.536,Z 283.993,A -85,B 0,C 180,E1 -8534.726,E2 -8534.726} C_VEL
LIN {X 0,Y 453.557,Z 283.987,A -85,B 0,C 180,E1 -8538.379,E2 -8538.379} C_VEL
LIN {X 0,Y 453.65,Z 283.974,A -85,B 0,C 180,E1 -8541.985,E2 -8541.985} C_VEL
LIN {X 0,Y 453.635,Z 283.979,A -85,B 0,C 180,E1 -8543.116,E2 -8543.116} C_VEL
LIN {X 0,Y 452.951,Z 284.062,A -85,B 0,C 180,E1 -8543.857,E2 -8543.857} C_VEL
LIN {X 0,Y 450.002,Z 284.432,A -85,B 0,C 180,E1 -8545.058,E2 -8545.058} C_VEL
LIN {X 0,Y 447.58,Z 284.731,A -85,B 0,C 180,E1 -8546.027,E2 -8546.027} C_VEL
LIN {X 0,Y 446.645,Z 284.851,A -85,B 0,C 180,E1 -8546.778,E2 -8546.778} C_VEL
LIN {X 0,Y 446.627,Z 284.849,A -85,B 0,C 180,E1 -8547.031,E2 -8547.031} C_VEL
LIN {X 0,Y 446.791,Z 284.828,A -85,B 0,C 180,E1 -8549.999,E2 -8549.999} C_VEL
LIN {X 0,Y 446.706,Z 284.842,A -85,B 0,C 180,E1 -8552.704,E2 -8552.704} C_VEL
LIN {X 0,Y 446.635,Z 284.848,A -85,B 0,C 180,E1 -8556.322,E2 -8556.322} C_VEL
LIN {X 0,Y 446.533,Z 284.865,A -85,B 0,C 180,E1 -8559.053,E2 -8559.053} C_VEL
LIN {X 0,Y 446.527,Z 284.864,A -85,B 0,C 180,E1 -8562.727,E2 -8562.727} C_VEL
LIN {X 0,Y 446.481,Z 284.867,A -85,B 0,C 180,E1 -8566.456,E2 -8566.456} C_VEL
LIN {X 0,Y 446.459,Z 284.873,A -85,B 0,C 180,E1 -8569.3,E2 -8569.3} C_VEL
LIN {X 0,Y 446.424,Z 284.873,A -85,B 0,C 180,E1 -8572.195,E2 -8572.195} C_VEL
LIN {X 0,Y 446.444,Z 284.877,A -85,B 0,C 180,E1 -8575.149,E2 -8575.149} C_VEL
LIN {X 0,Y 446.466,Z 284.867,A -85,B 0,C 180,E1 -8578.175,E2 -8578.175} C_VEL
LIN {X 0,Y 446.413,Z 284.879,A -85,B 0,C 180,E1 -8581.295,E2 -8581.295} C_VEL
LIN {X 0,Y 446.406,Z 284.875,A -85,B 0,C 180,E1 -8584.519,E2 -8584.519} C_VEL
LIN {X 0,Y 446.412,Z 284.874,A -85,B 0,C 180,E1 -8588.08,E2 -8588.08} C_VEL
LIN {X 0,Y 446.421,Z 284.879,A -85,B 0,C 180,E1 -8590.917,E2 -8590.917} C_VEL
LIN {X 0,Y 446.515,Z 284.898,A -85,B 0,C 180,E1 -8592.398,E2 -8592.398} C_VEL
LIN {X 0,Y 447.569,Z 291.86,A -85,B 0,C 180,E1 -8593.975,E2 -8593.975} C_VEL
LIN {X 0,Y 447.556,Z 293.466,A -85,B 0,C 180,E1 -8594.321,E2 -8594.321} C_VEL
LIN {X 0,Y 450.864,Z 309.739,A -85,B 0,C 180,E1 -8594.751,E2 -8594.751} C_VEL
LIN {X 0,Y 449.737,Z 401.186,A -85,B 0,C 180,E1 -8596.34,E2 -8596.34} C_VEL
LIN {X 0,Y 449.45,Z 414.811,A -85,B 0,C 180,E1 -8596.767,E2 -8596.767} C_VEL
LIN {X 0,Y 449.061,Z 427.407,A -85,B 0,C 180,E1 -8597.347,E2 -8597.347} C_VEL
LIN {X 0,Y 448.603,Z 439.507,A -85,B 0,C 180,E1 -8598.105,E2 -8598.105} C_VEL
LIN {X 0,Y 448.045,Z 450.662,A -85,B 0,C 180,E1 -8598.995,E2 -8598.995} C_VEL
LIN {X 0,Y 447.537,Z 461.143,A -85,B 0,C 180,E1 -8600.044,E2 -8600.044} C_VEL
LIN {X 0,Y 447.004,Z 470.92,A -85,B 0,C 180,E1 -8601.263,E2 -8601.263} C_VEL
LIN {X 0,Y 446.511,Z 480.175,A -85,B 0,C 180,E1 -8602.701,E2 -8602.701} C_VEL
LIN {X 0,Y 446.151,Z 487.332,A -85,B 0,C 180,E1 -8604.112,E2 -8604.112} C_VEL
LIN {X 0,Y 445.907,Z 492.688,A -85,B 0,C 180,E1 -8605.431,E2 -8605.431} C_VEL
LIN {X 0,Y 445.706,Z 497.955,A -85,B 0,C 180,E1 -8607.126,E2 -8607.126} C_VEL
LIN {X 0,Y 445.487,Z 501.216,A -85,B 0,C 180,E1 -8608.628,E2 -8608.628} C_VEL
LIN {X 0,Y 445.37,Z 503.36,A -85,B 0,C 180,E1 -8610.203,E2 -8610.203} C_VEL
LIN {X 0,Y 445.36,Z 504.329,A -85,B 0,C 180,E1 -8612.079,E2 -8612.079} C_VEL
LIN {X 0,Y 445.391,Z 503.658,A -85,B 0,C 180,E1 -8613.78,E2 -8613.78} C_VEL
LIN {X 0,Y 445.445,Z 502.603,A -85,B 0,C 180,E1 -8614.787,E2 -8614.787} C_VEL
LIN {X 0,Y 445.645,Z 500.343,A -85,B 0,C 180,E1 -8616.144,E2 -8616.144} C_VEL
LIN {X 0,Y 445.839,Z 496.361,A -85,B 0,C 180,E1 -8617.771,E2 -8617.771} C_VEL
LIN {X 0,Y 446.053,Z 491.39,A -85,B 0,C 180,E1 -8619.237,E2 -8619.237} C_VEL
LIN {X 0,Y 446.457,Z 484.489,A -85,B 0,C 180,E1 -8620.801,E2 -8620.801} C_VEL
LIN {X 0,Y 446.897,Z 477.006,A -85,B 0,C 180,E1 -8622.142,E2 -8622.142} C_VEL
LIN {X 0,Y 447.379,Z 468.544,A -85,B 0,C 180,E1 -8623.364,E2 -8623.364} C_VEL
LIN {X 0,Y 447.962,Z 458.566,A -85,B 0,C 180,E1 -8624.532,E2 -8624.532} C_VEL
LIN {X 0,Y 448.549,Z 448.529,A -85,B 0,C 180,E1 -8625.482,E2 -8625.482} C_VEL
LIN {X 0,Y 449.008,Z 437.326,A -85,B 0,C 180,E1 -8626.332,E2 -8626.332} C_VEL
LIN {X 0,Y 449.508,Z 424.622,A -85,B 0,C 180,E1 -8627.07,E2 -8627.07} C_VEL
LIN {X 0,Y 449.824,Z 412.313,A -85,B 0,C 180,E1 -8627.595,E2 -8627.595} C_VEL
LIN {X 0,Y 450.105,Z 399.705,A -85,B 0,C 180,E1 -8627.946,E2 -8627.946} C_VEL
LIN {X 0,Y 451.304,Z 309.284,A -85,B 0,C 180,E1 -8629.558,E2 -8629.558} C_VEL
LIN {X 0,Y 447.978,Z 293.292,A -85,B 0,C 180,E1 -8630.035,E2 -8630.035} C_VEL
LIN {X 0,Y 447.204,Z 287.979,A -85,B 0,C 180,E1 -8630.959,E2 -8630.959} C_VEL
LIN {X 0,Y 446.52,Z 284.865,A -85,B 0,C 180,E1 -8631.544,E2 -8631.544} C_VEL
LIN {X 0,Y 446.586,Z 284.861,A -85,B 0,C 180,E1 -8634.582,E2 -8634.582} C_VEL
LIN {X 0,Y 446.659,Z 284.851,A -85,B 0,C 180,E1 -8637.295,E2 -8637.295} C_VEL
LIN {X 0,Y 446.734,Z 284.836,A -85,B 0,C 180,E1 -8640,E2 -8640} C_VEL
LIN {X 0,Y 446.659,Z 284.849,A -85,B 0,C 180,E1 -8642.706,E2 -8642.706} C_VEL
LIN {X 0,Y 446.59,Z 284.854,A -85,B 0,C 180,E1 -8646.325,E2 -8646.325} C_VEL
LIN {X 0,Y 446.485,Z 284.872,A -85,B 0,C 180,E1 -8649.057,E2 -8649.057} C_VEL
LIN {X 0,Y 446.482,Z 284.869,A -85,B 0,C 180,E1 -8652.731,E2 -8652.731} C_VEL
LIN {X 0,Y 446.439,Z 284.872,A -85,B 0,C 180,E1 -8656.461,E2 -8656.461} C_VEL
LIN {X 0,Y 446.419,Z 284.876,A -85,B 0,C 180,E1 -8659.306,E2 -8659.306} C_VEL
LIN {X 0,Y 446.368,Z 284.88,A -85,B 0,C 180,E1 -8662.203,E2 -8662.203} C_VEL
LIN {X 0,Y 446.411,Z 284.878,A -85,B 0,C 180,E1 -8665.156,E2 -8665.156} C_VEL
LIN {X 0,Y 446.442,Z 284.87,A -85,B 0,C 180,E1 -8668.182,E2 -8668.182} C_VEL
LIN {X 0,Y 446.377,Z 284.878,A -85,B 0,C 180,E1 -8671.778,E2 -8671.778} C_VEL
LIN {X 0,Y 446.39,Z 284.876,A -85,B 0,C 180,E1 -8674.527,E2 -8674.527} C_VEL
LIN {X 0,Y 446.401,Z 284.876,A -85,B 0,C 180,E1 -8678.087,E2 -8678.087} C_VEL
LIN {X 0,Y 446.412,Z 284.878,A -85,B 0,C 180,E1 -8680.924,E2 -8680.924} C_VEL
LIN {X 0,Y 446.371,Z 284.881,A -85,B 0,C 180,E1 -8683.85,E2 -8683.85} C_VEL
LIN {X 0,Y 446.371,Z 284.88,A -85,B 0,C 180,E1 -8686.408,E2 -8686.408} C_VEL
LIN {X 0,Y 446.402,Z 284.88,A -85,B 0,C 180,E1 -8689.087,E2 -8689.087} C_VEL
LIN {X 0,Y 446.384,Z 284.879,A -85,B 0,C 180,E1 -8692.125,E2 -8692.125} C_VEL
LIN {X 0,Y 446.41,Z 284.885,A -85,B 0,C 180,E1 -8695.481,E2 -8695.481} C_VEL
LIN {X 0,Y 446.399,Z 284.885,A -85,B 0,C 180,E1 -8698.704,E2 -8698.704} C_VEL
LIN {X 0,Y 446.437,Z 284.878,A -85,B 0,C 180,E1 -8701.834,E2 -8701.834} C_VEL
LIN {X 0,Y 446.488,Z 284.972,A -85,B 0,C 180,E1 -8702.982,E2 -8702.982} C_VEL
LIN {X 0,Y 448.742,Z 296.138,A -85,B 0,C 180,E1 -8704.989,E2 -8704.989} C_VEL
LIN {X 0,Y 448.736,Z 303.534,A -85,B 0,C 180,E1 -8706.22,E2 -8706.22} C_VEL
LIN {X 0,Y 447.825,Z 325.488,A -85,B 0,C 180,E1 -8709.806,E2 -8709.806} C_VEL
LIN {X 0,Y 447.344,Z 339.197,A -85,B 0,C 180,E1 -8712.009,E2 -8712.009} C_VEL
LIN {X 0,Y 450.762,Z 363.36,A -85,B 0,C 180,E1 -8712.614,E2 -8712.614} C_VEL
LIN {X 0,Y 449.791,Z 449.02,A -85,B 0,C 180,E1 -8714.134,E2 -8714.134} C_VEL
LIN {X 0,Y 449.281,Z 462.719,A -85,B 0,C 180,E1 -8714.552,E2 -8714.552} C_VEL
LIN {X 0,Y 448.761,Z 475.727,A -85,B 0,C 180,E1 -8715.144,E2 -8715.144} C_VEL
LIN {X 0,Y 448.12,Z 488.402,A -85,B 0,C 180,E1 -8715.934,E2 -8715.934} C_VEL
LIN {X 0,Y 447.527,Z 499.52,A -85,B 0,C 180,E1 -8716.82,E2 -8716.82} C_VEL
LIN {X 0,Y 447.005,Z 509.999,A -85,B 0,C 180,E1 -8717.864,E2 -8717.864} C_VEL
LIN {X 0,Y 446.458,Z 520.1,A -85,B 0,C 180,E1 -8719.114,E2 -8719.114} C_VEL
LIN {X 0,Y 445.994,Z 529.009,A -85,B 0,C 180,E1 -8720.478,E2 -8720.478} C_VEL
LIN {X 0,Y 445.74,Z 536.126,A -85,B 0,C 180,E1 -8721.844,E2 -8721.844} C_VEL
LIN {X 0,Y 445.549,Z 542.012,A -85,B 0,C 180,E1 -8723.253,E2 -8723.253} C_VEL
LIN {X 0,Y 445.496,Z 546.34,A -85,B 0,C 180,E1 -8724.571,E2 -8724.571} C_VEL
LIN {X 0,Y 445.427,Z 548.721,A -85,B 0,C 180,E1 -8725.477,E2 -8725.477} C_VEL
LIN {X 0,Y 445.426,Z 550.653,A -85,B 0,C 180,E1 -8726.383,E2 -8726.383} C_VEL
LIN {X 0,Y 445.467,Z 552.105,A -85,B 0,C 180,E1 -8727.289,E2 -8727.289} C_VEL
LIN {X 0,Y 445.437,Z 553.146,A -85,B 0,C 180,E1 -8728.193,E2 -8728.193} C_VEL
LIN {X 0,Y 445.43,Z 553.787,A -85,B 0,C 180,E1 -8729.097,E2 -8729.097} C_VEL
LIN {X 0,Y 445.409,Z 554.005,A -85,B 0,C 180,E1 -8730.001,E2 -8730.001} C_VEL
LIN {X 0,Y 445.43,Z 553.783,A -85,B 0,C 180,E1 -8730.905,E2 -8730.905} C_VEL
LIN {X 0,Y 445.437,Z 553.162,A -85,B 0,C 180,E1 -8731.81,E2 -8731.81} C_VEL
LIN {X 0,Y 445.467,Z 552.141,A -85,B 0,C 180,E1 -8732.714,E2 -8732.714} C_VEL
LIN {X 0,Y 445.426,Z 550.669,A -85,B 0,C 180,E1 -8733.62,E2 -8733.62} C_VEL
LIN {X 0,Y 445.486,Z 547.632,A -85,B 0,C 180,E1 -8734.979,E2 -8734.979} C_VEL
LIN {X 0,Y 445.531,Z 543.339,A -85,B 0,C 180,E1 -8736.386,E2 -8736.386} C_VEL
LIN {X 0,Y 445.702,Z 537.153,A -85,B 0,C 180,E1 -8737.931,E2 -8737.931} C_VEL
LIN {X 0,Y 445.944,Z 530.225,A -85,B 0,C 180,E1 -8739.297,E2 -8739.297} C_VEL
LIN {X 0,Y 446.26,Z 523.151,A -85,B 0,C 180,E1 -8740.435,E2 -8740.435} C_VEL
LIN {X 0,Y 446.741,Z 514.632,A -85,B 0,C 180,E1 -8741.571,E2 -8741.571} C_VEL
LIN {X 0,Y 447.278,Z 504.099,A -85,B 0,C 180,E1 -8742.708,E2 -8742.708} C_VEL
LIN {X 0,Y 447.865,Z 492.25,A -85,B 0,C 180,E1 -8743.73,E2 -8743.73} C_VEL
LIN {X 0,Y 448.403,Z 480.385,A -85,B 0,C 180,E1 -8744.523,E2 -8744.523} C_VEL
LIN {X 0,Y 448.967,Z 466.824,A -85,B 0,C 180,E1 -8745.201,E2 -8745.201} C_VEL
LIN {X 0,Y 449.446,Z 453.652,A -85,B 0,C 180,E1 -8745.649,E2 -8745.649} C_VEL
LIN {X 0,Y 449.799,Z 436.551,A -85,B 0,C 180,E1 -8745.985,E2 -8745.985} C_VEL
LIN {X 0,Y 450.492,Z 363.553,A -85,B 0,C 180,E1 -8747.242,E2 -8747.242} C_VEL
LIN {X 0,Y 447.354,Z 341.226,A -85,B 0,C 180,E1 -8747.759,E2 -8747.759} C_VEL
LIN {X 0,Y 448.078,Z 324.284,A -85,B 0,C 180,E1 -8750.665,E2 -8750.665} C_VEL
LIN {X 0,Y 448.894,Z 309.16,A -85,B 0,C 180,E1 -8753.285,E2 -8753.285} C_VEL
LIN {X 0,Y 449.392,Z 299.522,A -85,B 0,C 180,E1 -8754.976,E2 -8754.976} C_VEL
LIN {X 0,Y 446.458,Z 284.873,A -85,B 0,C 180,E1 -8757.793,E2 -8757.793} C_VEL
LIN {X 0,Y 446.407,Z 284.877,A -85,B 0,C 180,E1 -8761.299,E2 -8761.299} C_VEL
LIN {X 0,Y 446.414,Z 284.88,A -85,B 0,C 180,E1 -8764.522,E2 -8764.522} C_VEL
LIN {X 0,Y 446.392,Z 284.878,A -85,B 0,C 180,E1 -8768.075,E2 -8768.075} C_VEL
LIN {X 0,Y 446.39,Z 284.878,A -85,B 0,C 180,E1 -8771.392,E2 -8771.392} C_VEL
LIN {X 0,Y 446.407,Z 284.878,A -85,B 0,C 180,E1 -8775.106,E2 -8775.106} C_VEL
LIN {X 0,Y 446.385,Z 284.883,A -85,B 0,C 180,E1 -8778.604,E2 -8778.604} C_VEL
LIN {X 0,Y 446.384,Z 284.879,A -85,B 0,C 180,E1 -8781.921,E2 -8781.921} C_VEL
LIN {X 0,Y 446.399,Z 284.877,A -85,B 0,C 180,E1 -8785.474,E2 -8785.474} C_VEL
LIN {X 0,Y 446.385,Z 284.883,A -85,B 0,C 180,E1 -8788.697,E2 -8788.697} C_VEL
LIN {X 0,Y 446.462,Z 284.869,A -85,B 0,C 180,E1 -8791.819,E2 -8791.819} C_VEL
LIN {X 0,Y 446.408,Z 284.881,A -85,B 0,C 180,E1 -8794.844,E2 -8794.844} C_VEL
LIN {X 0,Y 446.419,Z 284.876,A -85,B 0,C 180,E1 -8798.244,E2 -8798.244} C_VEL
LIN {X 0,Y 446.418,Z 284.875,A -85,B 0,C 180,E1 -8801.647,E2 -8801.647} C_VEL
LIN {X 0,Y 446.474,Z 284.87,A -85,B 0,C 180,E1 -8804.478,E2 -8804.478} C_VEL
LIN {X 0,Y 446.495,Z 284.867,A -85,B 0,C 180,E1 -8808.192,E2 -8808.192} C_VEL
LIN {X 0,Y 446.567,Z 284.857,A -85,B 0,C 180,E1 -8811.857,E2 -8811.857} C_VEL
LIN {X 0,Y 446.603,Z 284.854,A -85,B 0,C 180,E1 -8814.582,E2 -8814.582} C_VEL
LIN {X 0,Y 446.629,Z 284.851,A -85,B 0,C 180,E1 -8818.196,E2 -8818.196} C_VEL
LIN {X 0,Y 446.754,Z 284.834,A -85,B 0,C 180,E1 -8820,E2 -8820} C_VEL
LIN {X 0,Y 446.654,Z 284.848,A -85,B 0,C 180,E1 -8822.705,E2 -8822.705} C_VEL
LIN {X 0,Y 446.601,Z 284.855,A -85,B 0,C 180,E1 -8826.324,E2 -8826.324} C_VEL
LIN {X 0,Y 446.506,Z 284.868,A -85,B 0,C 180,E1 -8829.056,E2 -8829.056} C_VEL
LIN {X 0,Y 446.501,Z 284.867,A -85,B 0,C 180,E1 -8832.73,E2 -8832.73} C_VEL
LIN {X 0,Y 446.458,Z 284.873,A -85,B 0,C 180,E1 -8836.46,E2 -8836.46} C_VEL
LIN {X 0,Y 446.437,Z 284.876,A -85,B 0,C 180,E1 -8839.304,E2 -8839.304} C_VEL
LIN {X 0,Y 446.387,Z 284.881,A -85,B 0,C 180,E1 -8842.201,E2 -8842.201} C_VEL
LIN {X 0,Y 446.427,Z 284.877,A -85,B 0,C 180,E1 -8845.154,E2 -8845.154} C_VEL
LIN {X 0,Y 446.458,Z 284.872,A -85,B 0,C 180,E1 -8848.18,E2 -8848.18} C_VEL
LIN {X 0,Y 446.393,Z 284.882,A -85,B 0,C 180,E1 -8851.302,E2 -8851.302} C_VEL
LIN {X 0,Y 446.406,Z 284.88,A -85,B 0,C 180,E1 -8854.524,E2 -8854.524} C_VEL
LIN {X 0,Y 446.415,Z 284.877,A -85,B 0,C 180,E1 -8858.084,E2 -8858.084} C_VEL
LIN {X 0,Y 446.423,Z 284.877,A -85,B 0,C 180,E1 -8860.921,E2 -8860.921} C_VEL
LIN {X 0,Y 446.382,Z 284.88,A -85,B 0,C 180,E1 -8863.848,E2 -8863.848} C_VEL
LIN {X 0,Y 446.43,Z 284.876,A -85,B 0,C 180,E1 -8866.399,E2 -8866.399} C_VEL
LIN {X 0,Y 446.454,Z 284.872,A -85,B 0,C 180,E1 -8869.806,E2 -8869.806} C_VEL
LIN {X 0,Y 446.421,Z 284.876,A -85,B 0,C 180,E1 -8872.125,E2 -8872.125} C_VEL
LIN {X 0,Y 446.419,Z 284.878,A -85,B 0,C 180,E1 -8875.478,E2 -8875.478} C_VEL
LIN {X 0,Y 446.406,Z 284.881,A -85,B 0,C 180,E1 -8878.701,E2 -8878.701} C_VEL
LIN {X 0,Y 446.477,Z 284.869,A -85,B 0,C 180,E1 -8881.822,E2 -8881.822} C_VEL
LIN {X 0,Y 446.451,Z 284.875,A -85,B 0,C 180,E1 -8884.848,E2 -8884.848} C_VEL
LIN {X 0,Y 446.443,Z 284.873,A -85,B 0,C 180,E1 -8888.246,E2 -8888.246} C_VEL
LIN {X 0,Y 446.453,Z 284.872,A -85,B 0,C 180,E1 -8891.649,E2 -8891.649} C_VEL
LIN {X 0,Y 446.504,Z 284.866,A -85,B 0,C 180,E1 -8894.48,E2 -8894.48} C_VEL
LIN {X 0,Y 446.515,Z 284.863,A -85,B 0,C 180,E1 -8898.193,E2 -8898.193} C_VEL
LIN {X 0,Y 446.598,Z 284.853,A -85,B 0,C 180,E1 -8901.857,E2 -8901.857} C_VEL
LIN {X 0,Y 446.643,Z 284.849,A -85,B 0,C 180,E1 -8904.582,E2 -8904.582} C_VEL
LIN {X 0,Y 446.627,Z 284.849,A -85,B 0,C 180,E1 -8907.031,E2 -8907.031} C_VEL
LIN {X 0,Y 446.111,Z 284.917,A -85,B 0,C 180,E1 -8907.784,E2 -8907.784} C_VEL
LIN {X 0,Y 443.291,Z 285.275,A -85,B 0,C 180,E1 -8909.007,E2 -8909.007} C_VEL
LIN {X 0,Y 440.801,Z 285.586,A -85,B 0,C 180,E1 -8909.994,E2 -8909.994} C_VEL
LIN {X 0,Y 439.712,Z 285.717,A -85,B 0,C 180,E1 -8910.757,E2 -8910.757} C_VEL
LIN {X 0,Y 439.618,Z 285.726,A -85,B 0,C 180,E1 -8911.016,E2 -8911.016} C_VEL
LIN {X 0,Y 439.653,Z 285.721,A -85,B 0,C 180,E1 -8912.747,E2 -8912.747} C_VEL
LIN {X 0,Y 439.607,Z 285.724,A -85,B 0,C 180,E1 -8916.423,E2 -8916.423} C_VEL
LIN {X 0,Y 439.495,Z 285.74,A -85,B 0,C 180,E1 -8919.199,E2 -8919.199} C_VEL
LIN {X 0,Y 439.497,Z 285.74,A -85,B 0,C 180,E1 -8922.724,E2 -8922.724} C_VEL
LIN {X 0,Y 439.438,Z 285.744,A -85,B 0,C 180,E1 -8926.346,E2 -8926.346} C_VEL
LIN {X 0,Y 439.423,Z 285.746,A -85,B 0,C 180,E1 -8929.622,E2 -8929.622} C_VEL
LIN {X 0,Y 439.364,Z 285.754,A -85,B 0,C 180,E1 -8932.571,E2 -8932.571} C_VEL
LIN {X 0,Y 439.39,Z 285.751,A -85,B 0,C 180,E1 -8935.581,E2 -8935.581} C_VEL
LIN {X 0,Y 439.407,Z 285.749,A -85,B 0,C 180,E1 -8938.669,E2 -8938.669} C_VEL
LIN {X 0,Y 439.363,Z 285.752,A -85,B 0,C 180,E1 -8942.03,E2 -8942.03} C_VEL
LIN {X 0,Y 439.372,Z 285.756,A -85,B 0,C 180,E1 -8945.337,E2 -8945.337} C_VEL
LIN {X 0,Y 439.373,Z 285.752,A -85,B 0,C 180,E1 -8948.589,E2 -8948.589} C_VEL
LIN {X 0,Y 439.38,Z 285.756,A -85,B 0,C 180,E1 -8951.256,E2 -8951.256} C_VEL
LIN {X 0,Y 439.478,Z 285.909,A -85,B 0,C 180,E1 -8952.255,E2 -8952.255} C_VEL
LIN {X 0,Y 440.588,Z 292.016,A -85,B 0,C 180,E1 -8953.666,E2 -8953.666} C_VEL
LIN {X 0,Y 440.591,Z 293.868,A -85,B 0,C 180,E1 -8954.068,E2 -8954.068} C_VEL
LIN {X 0,Y 444.03,Z 310.95,A -85,B 0,C 180,E1 -8954.517,E2 -8954.517} C_VEL
LIN {X 0,Y 442.866,Z 401.628,A -85,B 0,C 180,E1 -8956.129,E2 -8956.129} C_VEL
LIN {X 0,Y 442.559,Z 415.234,A -85,B 0,C 180,E1 -8956.563,E2 -8956.563} C_VEL
LIN {X 0,Y 442.174,Z 427.118,A -85,B 0,C 180,E1 -8957.114,E2 -8957.114} C_VEL
LIN {X 0,Y 441.681,Z 439.771,A -85,B 0,C 180,E1 -8957.911,E2 -8957.911} C_VEL
LIN {X 0,Y 441.114,Z 450.79,A -85,B 0,C 180,E1 -8958.801,E2 -8958.801} C_VEL
LIN {X 0,Y 440.576,Z 461.239,A -85,B 0,C 180,E1 -8959.853,E2 -8959.853} C_VEL
LIN {X 0,Y 440.062,Z 470.676,A -85,B 0,C 180,E1 -8961.036,E2 -8961.036} C_VEL
LIN {X 0,Y 439.601,Z 478.918,A -85,B 0,C 180,E1 -8962.302,E2 -8962.302} C_VEL
LIN {X 0,Y 439.186,Z 486.284,A -85,B 0,C 180,E1 -8963.695,E2 -8963.695} C_VEL
LIN {X 0,Y 438.863,Z 493.08,A -85,B 0,C 180,E1 -8965.355,E2 -8965.355} C_VEL
LIN {X 0,Y 438.631,Z 498.131,A -85,B 0,C 180,E1 -8966.992,E2 -8966.992} C_VEL
LIN {X 0,Y 438.486,Z 500.744,A -85,B 0,C 180,E1 -8968.143,E2 -8968.143} C_VEL
LIN {X 0,Y 438.343,Z 502.483,A -85,B 0,C 180,E1 -8969.133,E2 -8969.133} C_VEL
LIN {X 0,Y 438.283,Z 503.753,A -85,B 0,C 180,E1 -8970.193,E2 -8970.193} C_VEL
LIN {X 0,Y 438.268,Z 504.684,A -85,B 0,C 180,E1 -8971.867,E2 -8971.867} C_VEL
LIN {X 0,Y 438.31,Z 504.029,A -85,B 0,C 180,E1 -8973.871,E2 -8973.871} C_VEL
LIN {X 0,Y 438.431,Z 502.269,A -85,B 0,C 180,E1 -8975.369,E2 -8975.369} C_VEL
LIN {X 0,Y 438.659,Z 499.33,A -85,B 0,C 180,E1 -8976.889,E2 -8976.889} C_VEL
LIN {X 0,Y 438.822,Z 495.23,A -85,B 0,C 180,E1 -8978.386,E2 -8978.386} C_VEL
LIN {X 0,Y 439.176,Z 489.808,A -85,B 0,C 180,E1 -8979.876,E2 -8979.876} C_VEL
LIN {X 0,Y 439.595,Z 482.875,A -85,B 0,C 180,E1 -8981.353,E2 -8981.353} C_VEL
LIN {X 0,Y 440.023,Z 475.627,A -85,B 0,C 180,E1 -8982.599,E2 -8982.599} C_VEL
LIN {X 0,Y 440.578,Z 467.153,A -85,B 0,C 180,E1 -8983.791,E2 -8983.791} C_VEL
LIN {X 0,Y 441.14,Z 457.713,A -85,B 0,C 180,E1 -8984.878,E2 -8984.878} C_VEL
LIN {X 0,Y 441.736,Z 447.513,A -85,B 0,C 180,E1 -8985.828,E2 -8985.828} C_VEL
LIN {X 0,Y 442.274,Z 436.09,A -85,B 0,C 180,E1 -8986.679,E2 -8986.679} C_VEL
LIN {X 0,Y 442.759,Z 423.644,A -85,B 0,C 180,E1 -8987.394,E2 -8987.394} C_VEL
LIN {X 0,Y 443.113,Z 410.569,A -85,B 0,C 180,E1 -8987.927,E2 -8987.927} C_VEL
LIN {X 0,Y 443.403,Z 396.745,A -85,B 0,C 180,E1 -8988.284,E2 -8988.284} C_VEL
LIN {X 0,Y 444.603,Z 310.048,A -85,B 0,C 180,E1 -8989.857,E2 -8989.857} C_VEL
LIN {X 0,Y 441.141,Z 293.839,A -85,B 0,C 180,E1 -8990.343,E2 -8990.343} C_VEL
LIN {X 0,Y 439.503,Z 285.74,A -85,B 0,C 180,E1 -8991.842,E2 -8991.842} C_VEL
LIN {X 0,Y 439.561,Z 285.736,A -85,B 0,C 180,E1 -8994.495,E2 -8994.495} C_VEL
LIN {X 0,Y 439.606,Z 285.73,A -85,B 0,C 180,E1 -8997.251,E2 -8997.251} C_VEL
LIN {X 0,Y 439.705,Z 285.712,A -85,B 0,C 180,E1 -9000,E2 -9000} C_VEL
LIN {X 0,Y 439.606,Z 285.727,A -85,B 0,C 180,E1 -9002.749,E2 -9002.749} C_VEL
LIN {X 0,Y 439.561,Z 285.731,A -85,B 0,C 180,E1 -9006.426,E2 -9006.426} C_VEL
LIN {X 0,Y 439.448,Z 285.748,A -85,B 0,C 180,E1 -9009.203,E2 -9009.203} C_VEL
LIN {X 0,Y 439.453,Z 285.744,A -85,B 0,C 180,E1 -9012.728,E2 -9012.728} C_VEL
LIN {X 0,Y 439.396,Z 285.749,A -85,B 0,C 180,E1 -9016.35,E2 -9016.35} C_VEL
LIN {X 0,Y 439.352,Z 285.753,A -85,B 0,C 180,E1 -9019.629,E2 -9019.629} C_VEL
LIN {X 0,Y 439.316,Z 285.76,A -85,B 0,C 180,E1 -9022.579,E2 -9022.579} C_VEL
LIN {X 0,Y 439.359,Z 285.752,A -85,B 0,C 180,E1 -9025.588,E2 -9025.588} C_VEL
LIN {X 0,Y 439.374,Z 285.753,A -85,B 0,C 180,E1 -9028.677,E2 -9028.677} C_VEL
LIN {X 0,Y 439.328,Z 285.755,A -85,B 0,C 180,E1 -9032.034,E2 -9032.034} C_VEL
LIN {X 0,Y 439.357,Z 285.759,A -85,B 0,C 180,E1 -9035.344,E2 -9035.344} C_VEL
LIN {X 0,Y 439.363,Z 285.754,A -85,B 0,C 180,E1 -9038.598,E2 -9038.598} C_VEL
LIN {X 0,Y 439.367,Z 285.758,A -85,B 0,C 180,E1 -9041.262,E2 -9041.262} C_VEL
LIN {X 0,Y 439.372,Z 285.753,A -85,B 0,C 180,E1 -9044.734,E2 -9044.734} C_VEL
LIN {X 0,Y 439.369,Z 285.755,A -85,B 0,C 180,E1 -9047.8,E2 -9047.8} C_VEL
LIN {X 0,Y 439.366,Z 285.753,A -85,B 0,C 180,E1 -9050.227,E2 -9050.227} C_VEL
LIN {X 0,Y 439.353,Z 285.76,A -85,B 0,C 180,E1 -9053.717,E2 -9053.717} C_VEL
LIN {X 0,Y 439.355,Z 285.764,A -85,B 0,C 180,E1 -9057.058,E2 -9057.058} C_VEL
LIN {X 0,Y 439.362,Z 285.759,A -85,B 0,C 180,E1 -9060.278,E2 -9060.278} C_VEL
LIN {X 0,Y 439.45,Z 285.887,A -85,B 0,C 180,E1 -9062.728,E2 -9062.728} C_VEL
LIN {X 0,Y 441.858,Z 297.614,A -85,B 0,C 180,E1 -9064.871,E2 -9064.871} C_VEL
LIN {X 0,Y 441.848,Z 304.729,A -85,B 0,C 180,E1 -9066.075,E2 -9066.075} C_VEL
LIN {X 0,Y 440.883,Z 326.568,A -85,B 0,C 180,E1 -9069.695,E2 -9069.695} C_VEL
LIN {X 0,Y 440.397,Z 338.573,A -85,B 0,C 180,E1 -9071.671,E2 -9071.671} C_VEL
LIN {X 0,Y 443.112,Z 356.968,A -85,B 0,C 180,E1 -9072.155,E2 -9072.155} C_VEL
LIN {X 0,Y 444.124,Z 365.548,A -85,B 0,C 180,E1 -9072.362,E2 -9072.362} C_VEL
LIN {X 0,Y 442.966,Z 449.054,A -85,B 0,C 180,E1 -9073.883,E2 -9073.883} C_VEL
LIN {X 0,Y 442.431,Z 463.297,A -85,B 0,C 180,E1 -9074.336,E2 -9074.336} C_VEL
LIN {X 0,Y 441.899,Z 475.465,A -85,B 0,C 180,E1 -9074.908,E2 -9074.908} C_VEL
LIN {X 0,Y 441.217,Z 488.104,A -85,B 0,C 180,E1 -9075.709,E2 -9075.709} C_VEL
LIN {X 0,Y 440.535,Z 500.159,A -85,B 0,C 180,E1 -9076.695,E2 -9076.695} C_VEL
LIN {X 0,Y 439.962,Z 510.653,A -85,B 0,C 180,E1 -9077.783,E2 -9077.783} C_VEL
LIN {X 0,Y 439.465,Z 519.757,A -85,B 0,C 180,E1 -9078.939,E2 -9078.939} C_VEL
LIN {X 0,Y 438.962,Z 528.658,A -85,B 0,C 180,E1 -9080.325,E2 -9080.325} C_VEL
LIN {X 0,Y 438.664,Z 535.767,A -85,B 0,C 180,E1 -9081.712,E2 -9081.712} C_VEL
LIN {X 0,Y 438.465,Z 541.474,A -85,B 0,C 180,E1 -9083.098,E2 -9083.098} C_VEL
LIN {X 0,Y 438.393,Z 545.96,A -85,B 0,C 180,E1 -9084.482,E2 -9084.482} C_VEL
LIN {X 0,Y 438.356,Z 548.339,A -85,B 0,C 180,E1 -9085.404,E2 -9085.404} C_VEL
LIN {X 0,Y 438.327,Z 550.265,A -85,B 0,C 180,E1 -9086.325,E2 -9086.325} C_VEL
LIN {X 0,Y 438.392,Z 551.717,A -85,B 0,C 180,E1 -9087.245,E2 -9087.245} C_VEL
LIN {X 0,Y 438.354,Z 552.755,A -85,B 0,C 180,E1 -9088.164,E2 -9088.164} C_VEL
LIN {X 0,Y 438.353,Z 553.394,A -85,B 0,C 180,E1 -9089.083,E2 -9089.083} C_VEL
LIN {X 0,Y 438.347,Z 553.606,A -85,B 0,C 180,E1 -9090.001,E2 -9090.001} C_VEL
LIN {X 0,Y 438.369,Z 553.381,A -85,B 0,C 180,E1 -9090.92,E2 -9090.92} C_VEL
LIN {X 0,Y 438.354,Z 552.753,A -85,B 0,C 180,E1 -9091.839,E2 -9091.839} C_VEL
LIN {X 0,Y 438.392,Z 551.726,A -85,B 0,C 180,E1 -9092.758,E2 -9092.758} C_VEL
LIN {X 0,Y 438.329,Z 550.24,A -85,B 0,C 180,E1 -9093.678,E2 -9093.678} C_VEL
LIN {X 0,Y 438.416,Z 547.188,A -85,B 0,C 180,E1 -9095.059,E2 -9095.059} C_VEL
LIN {X 0,Y 438.45,Z 543.039,A -85,B 0,C 180,E1 -9096.443,E2 -9096.443} C_VEL
LIN {X 0,Y 438.63,Z 536.663,A -85,B 0,C 180,E1 -9098.06,E2 -9098.06} C_VEL
LIN {X 0,Y 438.882,Z 529.708,A -85,B 0,C 180,E1 -9099.448,E2 -9099.448} C_VEL
LIN {X 0,Y 439.214,Z 522.602,A -85,B 0,C 180,E1 -9100.604,E2 -9100.604} C_VEL
LIN {X 0,Y 439.737,Z 514.037,A -85,B 0,C 180,E1 -9101.758,E2 -9101.758} C_VEL
LIN {X 0,Y 440.313,Z 503.432,A -85,B 0,C 180,E1 -9102.912,E2 -9102.912} C_VEL
LIN {X 0,Y 440.837,Z 492.943,A -85,B 0,C 180,E1 -9103.836,E2 -9103.836} C_VEL
LIN {X 0,Y 441.398,Z 481.455,A -85,B 0,C 180,E1 -9104.641,E2 -9104.641} C_VEL
LIN {X 0,Y 441.957,Z 468.344,A -85,B 0,C 180,E1 -9105.329,E2 -9105.329} C_VEL
LIN {X 0,Y 442.486,Z 455.275,A -85,B 0,C 180,E1 -9105.812,E2 -9105.812} C_VEL
LIN {X 0,Y 442.835,Z 441.25,A -85,B 0,C 180,E1 -9106.125,E2 -9106.125} C_VEL
LIN {X 0,Y 443.611,Z 363.894,A -85,B 0,C 180,E1 -9107.484,E2 -9107.484} C_VEL
LIN {X 0,Y 440.378,Z 340.717,A -85,B 0,C 180,E1 -9108.053,E2 -9108.053} C_VEL
LIN {X 0,Y 441.187,Z 323.814,A -85,B 0,C 180,E1 -9111.002,E2 -9111.002} C_VEL
LIN {X 0,Y 442.215,Z 305.938,A -85,B 0,C 180,E1 -9114.156,E2 -9114.156} C_VEL
LIN {X 0,Y 442.417,Z 300.59,A -85,B 0,C 180,E1 -9115.112,E2 -9115.112} C_VEL
LIN {X 0,Y 439.419,Z 285.752,A -85,B 0,C 180,E1 -9118.042,E2 -9118.042} C_VEL
LIN {X 0,Y 439.353,Z 285.76,A -85,B 0,C 180,E1 -9120.787,E2 -9120.787} C_VEL
LIN {X 0,Y 439.352,Z 285.756,A -85,B 0,C 180,E1 -9124.045,E2 -9124.045} C_VEL
LIN {X 0,Y 439.332,Z 285.761,A -85,B 0,C 180,E1 -9126.884,E2 -9126.884} C_VEL
LIN {X 0,Y 439.336,Z 285.756,A -85,B 0,C 180,E1 -9129.838,E2 -9129.838} C_VEL
LIN {X 0,Y 439.323,Z 285.763,A -85,B 0,C 180,E1 -9132.618,E2 -9132.618} C_VEL
LIN {X 0,Y 439.361,Z 285.754,A -85,B 0,C 180,E1 -9135.265,E2 -9135.265} C_VEL
LIN {X 0,Y 439.347,Z 285.761,A -85,B 0,C 180,E1 -9138.745,E2 -9138.745} C_VEL
LIN {X 0,Y 439.341,Z 285.756,A -85,B 0,C 180,E1 -9141.608,E2 -9141.608} C_VEL
LIN {X 0,Y 439.373,Z 285.758,A -85,B 0,C 180,E1 -9144.841,E2 -9144.841} C_VEL
LIN {X 0,Y 439.343,Z 285.757,A -85,B 0,C 180,E1 -9148.137,E2 -9148.137} C_VEL
LIN {X 0,Y 439.409,Z 285.748,A -85,B 0,C 180,E1 -9151.596,E2 -9151.596} C_VEL
LIN {X 0,Y 439.35,Z 285.757,A -85,B 0,C 180,E1 -9154.411,E2 -9154.411} C_VEL
LIN {X 0,Y 439.332,Z 285.758,A -85,B 0,C 180,E1 -9157.422,E2 -9157.422} C_VEL
LIN {X 0,Y 439.412,Z 285.75,A -85,B 0,C 180,E1 -9160.662,E2 -9160.662} C_VEL
LIN {X 0,Y 439.43,Z 285.746,A -85,B 0,C 180,E1 -9164.223,E2 -9164.223} C_VEL
LIN {X 0,Y 439.459,Z 285.743,A -85,B 0,C 180,E1 -9168,E2 -9168} C_VEL
LIN {X 0,Y 439.516,Z 285.735,A -85,B 0,C 180,E1 -9171.725,E2 -9171.725} C_VEL
LIN {X 0,Y 439.579,Z 285.728,A -85,B 0,C 180,E1 -9174.495,E2 -9174.495} C_VEL
LIN {X 0,Y 439.599,Z 285.726,A -85,B 0,C 180,E1 -9178.167,E2 -9178.167} C_VEL
LIN {X 0,Y 439.725,Z 285.71,A -85,B 0,C 180,E1 -9180,E2 -9180} C_VEL
LIN {X 0,Y 439.604,Z 285.726,A -85,B 0,C 180,E1 -9182.749,E2 -9182.749} C_VEL
LIN {X 0,Y 439.577,Z 285.729,A -85,B 0,C 180,E1 -9186.425,E2 -9186.425} C_VEL
LIN {X 0,Y 439.469,Z 285.745,A -85,B 0,C 180,E1 -9189.202,E2 -9189.202} C_VEL
LIN {X 0,Y 439.472,Z 285.742,A -85,B 0,C 180,E1 -9192.727,E2 -9192.727} C_VEL
LIN {X 0,Y 439.415,Z 285.75,A -85,B 0,C 180,E1 -9196.349,E2 -9196.349} C_VEL
LIN {X 0,Y 439.371,Z 285.754,A -85,B 0,C 180,E1 -9199.627,E2 -9199.627} C_VEL
LIN {X 0,Y 439.334,Z 285.76,A -85,B 0,C 180,E1 -9202.577,E2 -9202.577} C_VEL
LIN {X 0,Y 439.376,Z 285.754,A -85,B 0,C 180,E1 -9205.586,E2 -9205.586} C_VEL
LIN {X 0,Y 439.399,Z 285.752,A -85,B 0,C 180,E1 -9208.674,E2 -9208.674} C_VEL
LIN {X 0,Y 439.348,Z 285.757,A -85,B 0,C 180,E1 -9211.862,E2 -9211.862} C_VEL
LIN {X 0,Y 439.376,Z 285.755,A -85,B 0,C 180,E1 -9215.157,E2 -9215.157} C_VEL
LIN {X 0,Y 439.376,Z 285.755,A -85,B 0,C 180,E1 -9218.595,E2 -9218.595} C_VEL
LIN {X 0,Y 439.378,Z 285.755,A -85,B 0,C 180,E1 -9221.26,E2 -9221.26} C_VEL
LIN {X 0,Y 439.384,Z 285.754,A -85,B 0,C 180,E1 -9224.731,E2 -9224.731} C_VEL
LIN {X 0,Y 439.396,Z 285.751,A -85,B 0,C 180,E1 -9227.799,E2 -9227.799} C_VEL
LIN {X 0,Y 439.437,Z 285.746,A -85,B 0,C 180,E1 -9230.231,E2 -9230.231} C_VEL
LIN {X 0,Y 439.365,Z 285.755,A -85,B 0,C 180,E1 -9233.714,E2 -9233.714} C_VEL
LIN {X 0,Y 439.362,Z 285.756,A -85,B 0,C 180,E1 -9237.055,E2 -9237.055} C_VEL
LIN {X 0,Y 439.373,Z 285.754,A -85,B 0,C 180,E1 -9240.275,E2 -9240.275} C_VEL
LIN {X 0,Y 439.421,Z 285.748,A -85,B 0,C 180,E1 -9243.397,E2 -9243.397} C_VEL
LIN {X 0,Y 439.38,Z 285.754,A -85,B 0,C 180,E1 -9246.43,E2 -9246.43} C_VEL
LIN {X 0,Y 439.383,Z 285.753,A -85,B 0,C 180,E1 -9249.397,E2 -9249.397} C_VEL
LIN {X 0,Y 439.428,Z 285.747,A -85,B 0,C 180,E1 -9252.31,E2 -9252.31} C_VEL
LIN {X 0,Y 439.444,Z 285.746,A -85,B 0,C 180,E1 -9255.174,E2 -9255.174} C_VEL
LIN {X 0,Y 439.481,Z 285.74,A -85,B 0,C 180,E1 -9258.001,E2 -9258.001} C_VEL
LIN {X 0,Y 439.546,Z 285.732,A -85,B 0,C 180,E1 -9261.726,E2 -9261.726} C_VEL
LIN {X 0,Y 439.619,Z 285.724,A -85,B 0,C 180,E1 -9264.495,E2 -9264.495} C_VEL
LIN {X 0,Y 439.633,Z 285.72,A -85,B 0,C 180,E1 -9268.167,E2 -9268.167} C_VEL
LIN {X 0,Y 439.761,Z 285.704,A -85,B 0,C 180,E1 -9269.999,E2 -9269.999} C_VEL
LIN {X 0,Y 439.618,Z 285.726,A -85,B 0,C 180,E1 -9271.016,E2 -9271.016} C_VEL
LIN {X 0,Y 438.904,Z 285.812,A -85,B 0,C 180,E1 -9271.78,E2 -9271.78} C_VEL
LIN {X 0,Y 435.927,Z 286.186,A -85,B 0,C 180,E1 -9273.019,E2 -9273.019} C_VEL
LIN {X 0,Y 433.475,Z 286.491,A -85,B 0,C 180,E1 -9274.019,E2 -9274.019} C_VEL
LIN {X 0,Y 432.502,Z 286.612,A -85,B 0,C 180,E1 -9274.794,E2 -9274.794} C_VEL
LIN {X 0,Y 432.465,Z 286.613,A -85,B 0,C 180,E1 -9275.056,E2 -9275.056} C_VEL
LIN {X 0,Y 432.581,Z 286.599,A -85,B 0,C 180,E1 -9277.677,E2 -9277.677} C_VEL
LIN {X 0,Y 432.402,Z 286.623,A -85,B 0,C 180,E1 -9281.244,E2 -9281.244} C_VEL
LIN {X 0,Y 432.425,Z 286.622,A -85,B 0,C 180,E1 -9283.149,E2 -9283.149} C_VEL
LIN {X 0,Y 432.403,Z 286.621,A -85,B 0,C 180,E1 -9286.476,E2 -9286.476} C_VEL
LIN {X 0,Y 432.368,Z 286.625,A -85,B 0,C 180,E1 -9289.955,E2 -9289.955} C_VEL
LIN {X 0,Y 432.313,Z 286.636,A -85,B 0,C 180,E1 -9292.96,E2 -9292.96} C_VEL
LIN {X 0,Y 432.348,Z 286.627,A -85,B 0,C 180,E1 -9296.029,E2 -9296.029} C_VEL
LIN {X 0,Y 432.334,Z 286.634,A -85,B 0,C 180,E1 -9299.183,E2 -9299.183} C_VEL
LIN {X 0,Y 432.311,Z 286.631,A -85,B 0,C 180,E1 -9302.291,E2 -9302.291} C_VEL
LIN {X 0,Y 432.317,Z 286.632,A -85,B 0,C 180,E1 -9304.673,E2 -9304.673} C_VEL
LIN {X 0,Y 432.327,Z 286.628,A -85,B 0,C 180,E1 -9308.145,E2 -9308.145} C_VEL
LIN {X 0,Y 432.371,Z 286.629,A -85,B 0,C 180,E1 -9311.785,E2 -9311.785} C_VEL
LIN {X 0,Y 432.423,Z 286.838,A -85,B 0,C 180,E1 -9312.092,E2 -9312.092} C_VEL
LIN {X 0,Y 433.635,Z 294.148,A -85,B 0,C 180,E1 -9313.787,E2 -9313.787} C_VEL
LIN {X 0,Y 437.203,Z 312.069,A -85,B 0,C 180,E1 -9314.278,E2 -9314.278} C_VEL
LIN {X 0,Y 435.976,Z 402.388,A -85,B 0,C 180,E1 -9315.919,E2 -9315.919} C_VEL
LIN {X 0,Y 435.683,Z 415.868,A -85,B 0,C 180,E1 -9316.361,E2 -9316.361} C_VEL
LIN {X 0,Y 435.249,Z 428.21,A -85,B 0,C 180,E1 -9316.95,E2 -9316.95} C_VEL
LIN {X 0,Y 434.757,Z 440.107,A -85,B 0,C 180,E1 -9317.717,E2 -9317.717} C_VEL
LIN {X 0,Y 434.204,Z 450.665,A -85,B 0,C 180,E1 -9318.579,E2 -9318.579} C_VEL
LIN {X 0,Y 433.598,Z 461.544,A -85,B 0,C 180,E1 -9319.683,E2 -9319.683} C_VEL
LIN {X 0,Y 433.131,Z 469.998,A -85,B 0,C 180,E1 -9320.743,E2 -9320.743} C_VEL
LIN {X 0,Y 432.61,Z 479.028,A -85,B 0,C 180,E1 -9322.132,E2 -9322.132} C_VEL
LIN {X 0,Y 432.154,Z 486.646,A -85,B 0,C 180,E1 -9323.589,E2 -9323.589} C_VEL
LIN {X 0,Y 431.872,Z 491.933,A -85,B 0,C 180,E1 -9324.851,E2 -9324.851} C_VEL
LIN {X 0,Y 431.62,Z 497.017,A -85,B 0,C 180,E1 -9326.385,E2 -9326.385} C_VEL
LIN {X 0,Y 431.449,Z 500.687,A -85,B 0,C 180,E1 -9327.88,E2 -9327.88} C_VEL
LIN {X 0,Y 431.224,Z 503.673,A -85,B 0,C 180,E1 -9329.731,E2 -9329.731} C_VEL
LIN {X 0,Y 431.182,Z 504.61,A -85,B 0,C 180,E1 -9330.727,E2 -9330.727} C_VEL
LIN {X 0,Y 431.18,Z 505.065,A -85,B 0,C 180,E1 -9331.792,E2 -9331.792} C_VEL
LIN {X 0,Y 431.2,Z 505.042,A -85,B 0,C 180,E1 -9332.848,E2 -9332.848} C_VEL
LIN {X 0,Y 431.226,Z 504.458,A -85,B 0,C 180,E1 -9333.894,E2 -9333.894} C_VEL
LIN {X 0,Y 431.322,Z 503.397,A -85,B 0,C 180,E1 -9334.936,E2 -9334.936} C_VEL
LIN {X 0,Y 431.55,Z 500.846,A -85,B 0,C 180,E1 -9336.485,E2 -9336.485} C_VEL
LIN {X 0,Y 431.758,Z 496.927,A -85,B 0,C 180,E1 -9338.08,E2 -9338.08} C_VEL
LIN {X 0,Y 432.006,Z 492.131,A -85,B 0,C 180,E1 -9339.527,E2 -9339.527} C_VEL
LIN {X 0,Y 432.442,Z 485.713,A -85,B 0,C 180,E1 -9341.033,E2 -9341.033} C_VEL
LIN {X 0,Y 432.982,Z 477.682,A -85,B 0,C 180,E1 -9342.526,E2 -9342.526} C_VEL
LIN {X 0,Y 433.54,Z 469.23,A -85,B 0,C 180,E1 -9343.78,E2 -9343.78} C_VEL
LIN {X 0,Y 434.194,Z 459.184,A -85,B 0,C 180,E1 -9344.991,E2 -9344.991} C_VEL
LIN {X 0,Y 434.853,Z 449.105,A -85,B 0,C 180,E1 -9345.971,E2 -9345.971} C_VEL
LIN {X 0,Y 435.39,Z 438.198,A -85,B 0,C 180,E1 -9346.821,E2 -9346.821} C_VEL
LIN {X 0,Y 435.889,Z 426.215,A -85,B 0,C 180,E1 -9347.547,E2 -9347.547} C_VEL
LIN {X 0,Y 436.298,Z 413.407,A -85,B 0,C 180,E1 -9348.119,E2 -9348.119} C_VEL
LIN {X 0,Y 436.58,Z 401.172,A -85,B 0,C 180,E1 -9348.48,E2 -9348.48} C_VEL
LIN {X 0,Y 437.98,Z 311.152,A -85,B 0,C 180,E1 -9350.155,E2 -9350.155} C_VEL
LIN {X 0,Y 434.514,Z 295.569,A -85,B 0,C 180,E1 -9350.647,E2 -9350.647} C_VEL
LIN {X 0,Y 434.109,Z 294.193,A -85,B 0,C 180,E1 -9350.713,E2 -9350.713} C_VEL
LIN {X 0,Y 432.488,Z 286.615,A -85,B 0,C 180,E1 -9352.108,E2 -9352.108} C_VEL
LIN {X 0,Y 432.538,Z 286.611,A -85,B 0,C 180,E1 -9354.406,E2 -9354.406} C_VEL
LIN {X 0,Y 432.55,Z 286.607,A -85,B 0,C 180,E1 -9358.138,E2 -9358.138} C_VEL
LIN {X 0,Y 432.676,Z 286.587,A -85,B 0,C 180,E1 -9360,E2 -9360} C_VEL
LIN {X 0,Y 432.556,Z 286.606,A -85,B 0,C 180,E1 -9362.794,E2 -9362.794} C_VEL
LIN {X 0,Y 432.514,Z 286.609,A -85,B 0,C 180,E1 -9366.532,E2 -9366.532} C_VEL
LIN {X 0,Y 432.392,Z 286.625,A -85,B 0,C 180,E1 -9369.355,E2 -9369.355} C_VEL
LIN {X 0,Y 432.393,Z 286.624,A -85,B 0,C 180,E1 -9372.813,E2 -9372.813} C_VEL
LIN {X 0,Y 432.362,Z 286.626,A -85,B 0,C 180,E1 -9376.481,E2 -9376.481} C_VEL
LIN {X 0,Y 432.288,Z 286.631,A -85,B 0,C 180,E1 -9379.963,E2 -9379.963} C_VEL
LIN {X 0,Y 432.271,Z 286.638,A -85,B 0,C 180,E1 -9382.967,E2 -9382.967} C_VEL
LIN {X 0,Y 432.319,Z 286.627,A -85,B 0,C 180,E1 -9386.036,E2 -9386.036} C_VEL
LIN {X 0,Y 432.299,Z 286.635,A -85,B 0,C 180,E1 -9389.191,E2 -9389.191} C_VEL
LIN {X 0,Y 432.283,Z 286.634,A -85,B 0,C 180,E1 -9392.447,E2 -9392.447} C_VEL
LIN {X 0,Y 432.308,Z 286.634,A -85,B 0,C 180,E1 -9395.636,E2 -9395.636} C_VEL
LIN {X 0,Y 432.333,Z 286.631,A -85,B 0,C 180,E1 -9399.345,E2 -9399.345} C_VEL
LIN {X 0,Y 432.335,Z 286.627,A -85,B 0,C 180,E1 -9401.797,E2 -9401.797} C_VEL
LIN {X 0,Y 432.305,Z 286.632,A -85,B 0,C 180,E1 -9404.352,E2 -9404.352} C_VEL
LIN {X 0,Y 432.294,Z 286.637,A -85,B 0,C 180,E1 -9407.02,E2 -9407.02} C_VEL
LIN {X 0,Y 432.31,Z 286.634,A -85,B 0,C 180,E1 -9409.825,E2 -9409.825} C_VEL
LIN {X 0,Y 432.284,Z 286.64,A -85,B 0,C 180,E1 -9413.026,E2 -9413.026} C_VEL
LIN {X 0,Y 432.341,Z 286.635,A -85,B 0,C 180,E1 -9416.001,E2 -9416.001} C_VEL
LIN {X 0,Y 432.331,Z 286.64,A -85,B 0,C 180,E1 -9419.494,E2 -9419.494} C_VEL
LIN {X 0,Y 432.353,Z 286.687,A -85,B 0,C 180,E1 -9422.439,E2 -9422.439} C_VEL
LIN {X 0,Y 434.989,Z 299.318,A -85,B 0,C 180,E1 -9424.794,E2 -9424.794} C_VEL
LIN {X 0,Y 434.955,Z 305.925,A -85,B 0,C 180,E1 -9425.926,E2 -9425.926} C_VEL
LIN {X 0,Y 433.914,Z 327.956,A -85,B 0,C 180,E1 -9429.625,E2 -9429.625} C_VEL
LIN {X 0,Y 433.508,Z 338.068,A -85,B 0,C 180,E1 -9431.32,E2 -9431.32} C_VEL
LIN {X 0,Y 436.375,Z 357.117,A -85,B 0,C 180,E1 -9431.846,E2 -9431.846} C_VEL
LIN {X 0,Y 437.413,Z 366.693,A -85,B 0,C 180,E1 -9432.079,E2 -9432.079} C_VEL
LIN {X 0,Y 436.229,Z 448.355,A -85,B 0,C 180,E1 -9433.597,E2 -9433.597} C_VEL
LIN {X 0,Y 435.676,Z 461.903,A -85,B 0,C 180,E1 -9434.027,E2 -9434.027} C_VEL
LIN {X 0,Y 435.098,Z 474.311,A -85,B 0,C 180,E1 -9434.606,E2 -9434.606} C_VEL
LIN {X 0,Y 434.427,Z 486.291,A -85,B 0,C 180,E1 -9435.361,E2 -9435.361} C_VEL
LIN {X 0,Y 433.712,Z 497.822,A -85,B 0,C 180,E1 -9436.292,E2 -9436.292} C_VEL
LIN {X 0,Y 433.066,Z 508.303,A -85,B 0,C 180,E1 -9437.348,E2 -9437.348} C_VEL
LIN {X 0,Y 432.573,Z 517.746,A -85,B 0,C 180,E1 -9438.523,E2 -9438.523} C_VEL
LIN {X 0,Y 431.965,Z 526.935,A -85,B 0,C 180,E1 -9439.93,E2 -9439.93} C_VEL
LIN {X 0,Y 431.649,Z 534.353,A -85,B 0,C 180,E1 -9441.34,E2 -9441.34} C_VEL
LIN {X 0,Y 431.431,Z 539.363,A -85,B 0,C 180,E1 -9442.514,E2 -9442.514} C_VEL
LIN {X 0,Y 431.286,Z 544.545,A -85,B 0,C 180,E1 -9444.019,E2 -9444.019} C_VEL
LIN {X 0,Y 431.287,Z 547.973,A -85,B 0,C 180,E1 -9445.328,E2 -9445.328} C_VEL
LIN {X 0,Y 431.23,Z 549.888,A -85,B 0,C 180,E1 -9446.264,E2 -9446.264} C_VEL
LIN {X 0,Y 431.318,Z 551.336,A -85,B 0,C 180,E1 -9447.2,E2 -9447.2} C_VEL
LIN {X 0,Y 431.274,Z 552.369,A -85,B 0,C 180,E1 -9448.134,E2 -9448.134} C_VEL
LIN {X 0,Y 431.264,Z 553.005,A -85,B 0,C 180,E1 -9449.068,E2 -9449.068} C_VEL
LIN {X 0,Y 431.286,Z 553.204,A -85,B 0,C 180,E1 -9450.001,E2 -9450.001} C_VEL
LIN {X 0,Y 431.279,Z 552.97,A -85,B 0,C 180,E1 -9450.935,E2 -9450.935} C_VEL
LIN {X 0,Y 431.274,Z 552.336,A -85,B 0,C 180,E1 -9451.869,E2 -9451.869} C_VEL
LIN {X 0,Y 431.319,Z 551.302,A -85,B 0,C 180,E1 -9452.803,E2 -9452.803} C_VEL
LIN {X 0,Y 431.234,Z 549.795,A -85,B 0,C 180,E1 -9453.739,E2 -9453.739} C_VEL
LIN {X 0,Y 431.322,Z 546.721,A -85,B 0,C 180,E1 -9455.143,E2 -9455.143} C_VEL
LIN {X 0,Y 431.378,Z 542.546,A -85,B 0,C 180,E1 -9456.549,E2 -9456.549} C_VEL
LIN {X 0,Y 431.572,Z 536.136,A -85,B 0,C 180,E1 -9458.193,E2 -9458.193} C_VEL
LIN {X 0,Y 431.842,Z 529.138,A -85,B 0,C 180,E1 -9459.603,E2 -9459.603} C_VEL
LIN {X 0,Y 432.199,Z 521.985,A -85,B 0,C 180,E1 -9460.778,E2 -9460.778} C_VEL
LIN {X 0,Y 432.715,Z 513.342,A -85,B 0,C 180,E1 -9461.952,E2 -9461.952} C_VEL
LIN {X 0,Y 433.335,Z 502.666,A -85,B 0,C 180,E1 -9463.124,E2 -9463.124} C_VEL
LIN {X 0,Y 433.896,Z 492.095,A -85,B 0,C 180,E1 -9464.061,E2 -9464.061} C_VEL
LIN {X 0,Y 434.476,Z 480.448,A -85,B 0,C 180,E1 -9464.88,E2 -9464.88} C_VEL
LIN {X 0,Y 435.02,Z 468.418,A -85,B 0,C 180,E1 -9465.52,E2 -9465.52} C_VEL
LIN {X 0,Y 435.551,Z 455.538,A -85,B 0,C 180,E1 -9466.011,E2 -9466.011} C_VEL
LIN {X 0,Y 435.927,Z 442.112,A -85,B 0,C 180,E1 -9466.327,E2 -9466.327} C_VEL
LIN {X 0,Y 436.79,Z 364.95,A -85,B 0,C 180,E1 -9467.709,E2 -9467.709} C_VEL
LIN {X 0,Y 433.443,Z 340.401,A -85,B 0,C 180,E1 -9468.322,E2 -9468.322} C_VEL
LIN {X 0,Y 434.453,Z 320.57,A -85,B 0,C 180,E1 -9471.842,E2 -9471.842} C_VEL
LIN {X 0,Y 435.476,Z 304.063,A -85,B 0,C 180,E1 -9474.809,E2 -9474.809} C_VEL
LIN {X 0,Y 435.173,Z 300.323,A -85,B 0,C 180,E1 -9475.514,E2 -9475.514} C_VEL
LIN {X 0,Y 432.391,Z 286.626,A -85,B 0,C 180,E1 -9478.249,E2 -9478.249} C_VEL
LIN {X 0,Y 432.313,Z 286.633,A -85,B 0,C 180,E1 -9481.345,E2 -9481.345} C_VEL
LIN {X 0,Y 432.32,Z 286.637,A -85,B 0,C 180,E1 -9484.677,E2 -9484.677} C_VEL
LIN {X 0,Y 432.315,Z 286.632,A -85,B 0,C 180,E1 -9488.15,E2 -9488.15} C_VEL
LIN {X 0,Y 432.293,Z 286.633,A -85,B 0,C 180,E1 -9491.799,E2 -9491.799} C_VEL
LIN {X 0,Y 432.319,Z 286.632,A -85,B 0,C 180,E1 -9494.346,E2 -9494.346} C_VEL
LIN {X 0,Y 432.289,Z 286.638,A -85,B 0,C 180,E1 -9497.016,E2 -9497.016} C_VEL
LIN {X 0,Y 432.272,Z 286.637,A -85,B 0,C 180,E1 -9499.826,E2 -9499.826} C_VEL
LIN {X 0,Y 432.282,Z 286.639,A -85,B 0,C 180,E1 -9503.019,E2 -9503.019} C_VEL
LIN {X 0,Y 432.312,Z 286.632,A -85,B 0,C 180,E1 -9506,E2 -9506} C_VEL
LIN {X 0,Y 432.318,Z 286.632,A -85,B 0,C 180,E1 -9509.489,E2 -9509.489} C_VEL
LIN {X 0,Y 432.347,Z 286.628,A -85,B 0,C 180,E1 -9511.874,E2 -9511.874} C_VEL
LIN {X 0,Y 432.339,Z 286.629,A -85,B 0,C 180,E1 -9515.541,E2 -9515.541} C_VEL
LIN {X 0,Y 432.319,Z 286.635,A -85,B 0,C 180,E1 -9519.044,E2 -9519.044} C_VEL
LIN {X 0,Y 432.328,Z 286.631,A -85,B 0,C 180,E1 -9522.009,E2 -9522.009} C_VEL
LIN {X 0,Y 432.361,Z 286.631,A -85,B 0,C 180,E1 -9524.925,E2 -9524.925} C_VEL
LIN {X 0,Y 432.433,Z 286.618,A -85,B 0,C 180,E1 -9527.802,E2 -9527.802} C_VEL
LIN {X 0,Y 432.46,Z 286.615,A -85,B 0,C 180,E1 -9531.589,E2 -9531.589} C_VEL
LIN {X 0,Y 432.556,Z 286.603,A -85,B 0,C 180,E1 -9534.405,E2 -9534.405} C_VEL
LIN {X 0,Y 432.569,Z 286.602,A -85,B 0,C 180,E1 -9538.137,E2 -9538.137} C_VEL
LIN {X 0,Y 432.695,Z 286.586,A -85,B 0,C 180,E1 -9540,E2 -9540} C_VEL
LIN {X 0,Y 432.556,Z 286.604,A -85,B 0,C 180,E1 -9542.793,E2 -9542.793} C_VEL
LIN {X 0,Y 432.533,Z 286.606,A -85,B 0,C 180,E1 -9546.53,E2 -9546.53} C_VEL
LIN {X 0,Y 432.412,Z 286.623,A -85,B 0,C 180,E1 -9549.353,E2 -9549.353} C_VEL
LIN {X 0,Y 432.413,Z 286.621,A -85,B 0,C 180,E1 -9552.811,E2 -9552.811} C_VEL
LIN {X 0,Y 432.381,Z 286.626,A -85,B 0,C 180,E1 -9556.479,E2 -9556.479} C_VEL
LIN {X 0,Y 432.307,Z 286.634,A -85,B 0,C 180,E1 -9559.961,E2 -9559.961} C_VEL
LIN {X 0,Y 432.289,Z 286.637,A -85,B 0,C 180,E1 -9562.965,E2 -9562.965} C_VEL
LIN {X 0,Y 432.336,Z 286.631,A -85,B 0,C 180,E1 -9566.034,E2 -9566.034} C_VEL
LIN {X 0,Y 432.326,Z 286.633,A -85,B 0,C 180,E1 -9569.188,E2 -9569.188} C_VEL
LIN {X 0,Y 432.3,Z 286.636,A -85,B 0,C 180,E1 -9572.294,E2 -9572.294} C_VEL
LIN {X 0,Y 432.317,Z 286.634,A -85,B 0,C 180,E1 -9574.679,E2 -9574.679} C_VEL
LIN {X 0,Y 432.33,Z 286.632,A -85,B 0,C 180,E1 -9578.15,E2 -9578.15} C_VEL
LIN {X 0,Y 432.347,Z 286.63,A -85,B 0,C 180,E1 -9581.608,E2 -9581.608} C_VEL
LIN {X 0,Y 432.317,Z 286.634,A -85,B 0,C 180,E1 -9584.349,E2 -9584.349} C_VEL
LIN {X 0,Y 432.35,Z 286.629,A -85,B 0,C 180,E1 -9587.011,E2 -9587.011} C_VEL
LIN {X 0,Y 432.344,Z 286.63,A -85,B 0,C 180,E1 -9589.818,E2 -9589.818} C_VEL
LIN {X 0,Y 432.305,Z 286.635,A -85,B 0,C 180,E1 -9593.024,E2 -9593.024} C_VEL
LIN {X 0,Y 432.349,Z 286.629,A -85,B 0,C 180,E1 -9595.998,E2 -9595.998} C_VEL
LIN {X 0,Y 432.338,Z 286.631,A -85,B 0,C 180,E1 -9599.491,E2 -9599.491} C_VEL
LIN {X 0,Y 432.384,Z 286.626,A -85,B 0,C 180,E1 -9602.929,E2 -9602.929} C_VEL
LIN {X 0,Y 432.365,Z 286.627,A -85,B 0,C 180,E1 -9606.024,E2 -9606.024} C_VEL
LIN {X 0,Y 432.345,Z 286.63,A -85,B 0,C 180,E1 -9609.046,E2 -9609.046} C_VEL
LIN {X 0,Y 432.374,Z 286.625,A -85,B 0,C 180,E1 -9612.011,E2 -9612.011} C_VEL
LIN {X 0,Y 432.392,Z 286.626,A -85,B 0,C 180,E1 -9614.926,E2 -9614.926} C_VEL
LIN {X 0,Y 432.456,Z 286.615,A -85,B 0,C 180,E1 -9617.803,E2 -9617.803} C_VEL
LIN {X 0,Y 432.49,Z 286.611,A -85,B 0,C 180,E1 -9621.59,E2 -9621.59} C_VEL
LIN {X 0,Y 432.595,Z 286.598,A -85,B 0,C 180,E1 -9624.405,E2 -9624.405} C_VEL
LIN {X 0,Y 432.603,Z 286.596,A -85,B 0,C 180,E1 -9628.137,E2 -9628.137} C_VEL
LIN {X 0,Y 432.731,Z 286.58,A -85,B 0,C 180,E1 -9629.999,E2 -9629.999} C_VEL
LIN {X 0,Y 432.602,Z 286.6,A -85,B 0,C 180,E1 -9632.792,E2 -9632.792} C_VEL
LIN {X 0,Y 432.465,Z 286.613,A -85,B 0,C 180,E1 -9635.056,E2 -9635.056} C_VEL
LIN {X 0,Y 431.904,Z 286.683,A -85,B 0,C 180,E1 -9635.835,E2 -9635.835} C_VEL
LIN {X 0,Y 429.054,Z 287.042,A -85,B 0,C 180,E1 -9637.099,E2 -9637.099} C_VEL
LIN {X 0,Y 426.567,Z 287.349,A -85,B 0,C 180,E1 -9638.12,E2 -9638.12} C_VEL
LIN {X 0,Y 425.488,Z 287.487,A -85,B 0,C 180,E1 -9638.91,E2 -9638.91} C_VEL
LIN {X 0,Y 425.398,Z 287.493,A -85,B 0,C 180,E1 -9639.178,E2 -9639.178} C_VEL
LIN {X 0,Y 425.397,Z 287.498,A -85,B 0,C 180,E1 -9642.908,E2 -9642.908} C_VEL
LIN {X 0,Y 425.352,Z 287.5,A -85,B 0,C 180,E1 -9646.602,E2 -9646.602} C_VEL
LIN {X 0,Y 425.351,Z 287.499,A -85,B 0,C 180,E1 -9649.645,E2 -9649.645} C_VEL
LIN {X 0,Y 425.298,Z 287.508,A -85,B 0,C 180,E1 -9653.361,E2 -9653.361} C_VEL
LIN {X 0,Y 425.332,Z 287.504,A -85,B 0,C 180,E1 -9656.841,E2 -9656.841} C_VEL
LIN {X 0,Y 425.3,Z 287.505,A -85,B 0,C 180,E1 -9659.714,E2 -9659.714} C_VEL
LIN {X 0,Y 425.263,Z 287.515,A -85,B 0,C 180,E1 -9663.044,E2 -9663.044} C_VEL
LIN {X 0,Y 425.26,Z 287.509,A -85,B 0,C 180,E1 -9665.925,E2 -9665.925} C_VEL
LIN {X 0,Y 425.288,Z 287.511,A -85,B 0,C 180,E1 -9669.043,E2 -9669.043} C_VEL
LIN {X 0,Y 425.344,Z 287.615,A -85,B 0,C 180,E1 -9671.888,E2 -9671.888} C_VEL
LIN {X 0,Y 426.635,Z 294.495,A -85,B 0,C 180,E1 -9673.511,E2 -9673.511} C_VEL
LIN {X 0,Y 430.353,Z 312.148,A -85,B 0,C 180,E1 -9674.011,E2 -9674.011} C_VEL
LIN {X 0,Y 429.136,Z 402.113,A -85,B 0,C 180,E1 -9675.675,E2 -9675.675} C_VEL
LIN {X 0,Y 428.808,Z 415.783,A -85,B 0,C 180,E1 -9676.123,E2 -9676.123} C_VEL
LIN {X 0,Y 428.321,Z 428.95,A -85,B 0,C 180,E1 -9676.762,E2 -9676.762} C_VEL
LIN {X 0,Y 427.835,Z 440.27,A -85,B 0,C 180,E1 -9677.503,E2 -9677.503} C_VEL
LIN {X 0,Y 427.251,Z 450.933,A -85,B 0,C 180,E1 -9678.384,E2 -9678.384} C_VEL
LIN {X 0,Y 426.681,Z 461.447,A -85,B 0,C 180,E1 -9679.463,E2 -9679.463} C_VEL
LIN {X 0,Y 426.082,Z 471.116,A -85,B 0,C 180,E1 -9680.699,E2 -9680.699} C_VEL
LIN {X 0,Y 425.569,Z 479.607,A -85,B 0,C 180,E1 -9682.037,E2 -9682.037} C_VEL
LIN {X 0,Y 425.124,Z 487.009,A -85,B 0,C 180,E1 -9683.478,E2 -9683.478} C_VEL
LIN {X 0,Y 424.795,Z 492.848,A -85,B 0,C 180,E1 -9684.907,E2 -9684.907} C_VEL
LIN {X 0,Y 424.539,Z 497.512,A -85,B 0,C 180,E1 -9686.362,E2 -9686.362} C_VEL
LIN {X 0,Y 424.346,Z 501.382,A -85,B 0,C 180,E1 -9687.996,E2 -9687.996} C_VEL
LIN {X 0,Y 424.151,Z 503.78,A -85,B 0,C 180,E1 -9689.486,E2 -9689.486} C_VEL
LIN {X 0,Y 424.107,Z 505.38,A -85,B 0,C 180,E1 -9691.421,E2 -9691.421} C_VEL
LIN {X 0,Y 424.089,Z 505.517,A -85,B 0,C 180,E1 -9692.354,E2 -9692.354} C_VEL
LIN {X 0,Y 424.135,Z 505.185,A -85,B 0,C 180,E1 -9693.466,E2 -9693.466} C_VEL
LIN {X 0,Y 424.202,Z 504.405,A -85,B 0,C 180,E1 -9694.485,E2 -9694.485} C_VEL
LIN {X 0,Y 424.314,Z 502.932,A -85,B 0,C 180,E1 -9695.624,E2 -9695.624} C_VEL
LIN {X 0,Y 424.56,Z 500.114,A -85,B 0,C 180,E1 -9697.108,E2 -9697.108} C_VEL
LIN {X 0,Y 424.756,Z 496.01,A -85,B 0,C 180,E1 -9698.654,E2 -9698.654} C_VEL
LIN {X 0,Y 425.214,Z 489.757,A -85,B 0,C 180,E1 -9700.387,E2 -9700.387} C_VEL
LIN {X 0,Y 425.741,Z 482.327,A -85,B 0,C 180,E1 -9701.97,E2 -9701.97} C_VEL
LIN {X 0,Y 426.339,Z 474.143,A -85,B 0,C 180,E1 -9703.352,E2 -9703.352} C_VEL
LIN {X 0,Y 426.974,Z 464.913,A -85,B 0,C 180,E1 -9704.609,E2 -9704.609} C_VEL
LIN {X 0,Y 427.706,Z 454.27,A -85,B 0,C 180,E1 -9705.779,E2 -9705.779} C_VEL
LIN {X 0,Y 428.347,Z 443.483,A -85,B 0,C 180,E1 -9706.721,E2 -9706.721} C_VEL
LIN {X 0,Y 428.97,Z 430.847,A -85,B 0,C 180,E1 -9707.583,E2 -9707.583} C_VEL
LIN {X 0,Y 429.384,Z 418.946,A -85,B 0,C 180,E1 -9708.195,E2 -9708.195} C_VEL
LIN {X 0,Y 429.725,Z 406.052,A -85,B 0,C 180,E1 -9708.653,E2 -9708.653} C_VEL
LIN {X 0,Y 430.114,Z 383.968,A -85,B 0,C 180,E1 -9709.108,E2 -9709.108} C_VEL
LIN {X 0,Y 431.38,Z 312.367,A -85,B 0,C 180,E1 -9710.472,E2 -9710.472} C_VEL
LIN {X 0,Y 428.066,Z 297.473,A -85,B 0,C 180,E1 -9710.953,E2 -9710.953} C_VEL
LIN {X 0,Y 427.017,Z 294.594,A -85,B 0,C 180,E1 -9711.095,E2 -9711.095} C_VEL
LIN {X 0,Y 425.468,Z 287.49,A -85,B 0,C 180,E1 -9712.455,E2 -9712.455} C_VEL
LIN {X 0,Y 425.494,Z 287.488,A -85,B 0,C 180,E1 -9714.313,E2 -9714.313} C_VEL
LIN {X 0,Y 425.52,Z 287.483,A -85,B 0,C 180,E1 -9718.108,E2 -9718.108} C_VEL
LIN {X 0,Y 425.646,Z 287.463,A -85,B 0,C 180,E1 -9720,E2 -9720} C_VEL
LIN {X 0,Y 425.508,Z 287.483,A -85,B 0,C 180,E1 -9722.841,E2 -9722.841} C_VEL
LIN {X 0,Y 425.472,Z 287.486,A -85,B 0,C 180,E1 -9726.64,E2 -9726.64} C_VEL
LIN {X 0,Y 425.352,Z 287.5,A -85,B 0,C 180,E1 -9729.511,E2 -9729.511} C_VEL
LIN {X 0,Y 425.353,Z 287.501,A -85,B 0,C 180,E1 -9732.912,E2 -9732.912} C_VEL
LIN {X 0,Y 425.311,Z 287.506,A -85,B 0,C 180,E1 -9736.607,E2 -9736.607} C_VEL
LIN {X 0,Y 425.279,Z 287.506,A -85,B 0,C 180,E1 -9739.638,E2 -9739.638} C_VEL
LIN {X 0,Y 425.259,Z 287.511,A -85,B 0,C 180,E1 -9743.368,E2 -9743.368} C_VEL
LIN {X 0,Y 425.304,Z 287.505,A -85,B 0,C 180,E1 -9746.847,E2 -9746.847} C_VEL
LIN {X 0,Y 425.248,Z 287.513,A -85,B 0,C 180,E1 -9749.723,E2 -9749.723} C_VEL
LIN {X 0,Y 425.243,Z 287.516,A -85,B 0,C 180,E1 -9753.052,E2 -9753.052} C_VEL
LIN {X 0,Y 425.247,Z 287.512,A -85,B 0,C 180,E1 -9755.933,E2 -9755.933} C_VEL
LIN {X 0,Y 425.279,Z 287.512,A -85,B 0,C 180,E1 -9759.05,E2 -9759.05} C_VEL
LIN {X 0,Y 425.285,Z 287.505,A -85,B 0,C 180,E1 -9761.966,E2 -9761.966} C_VEL
LIN {X 0,Y 425.257,Z 287.515,A -85,B 0,C 180,E1 -9765.287,E2 -9765.287} C_VEL
LIN {X 0,Y 425.249,Z 287.513,A -85,B 0,C 180,E1 -9768.625,E2 -9768.625} C_VEL
LIN {X 0,Y 425.27,Z 287.513,A -85,B 0,C 180,E1 -9771.105,E2 -9771.105} C_VEL
LIN {X 0,Y 425.28,Z 287.512,A -85,B 0,C 180,E1 -9774.668,E2 -9774.668} C_VEL
LIN {X 0,Y 425.248,Z 287.521,A -85,B 0,C 180,E1 -9778.077,E2 -9778.077} C_VEL
LIN {X 0,Y 425.301,Z 287.512,A -85,B 0,C 180,E1 -9781.371,E2 -9781.371} C_VEL
LIN {X 0,Y 425.323,Z 287.657,A -85,B 0,C 180,E1 -9782.145,E2 -9782.145} C_VEL
LIN {X 0,Y 428.018,Z 300.294,A -85,B 0,C 180,E1 -9784.569,E2 -9784.569} C_VEL
LIN {X 0,Y 428.095,Z 305.68,A -85,B 0,C 180,E1 -9785.515,E2 -9785.515} C_VEL
LIN {X 0,Y 427.094,Z 326.211,A -85,B 0,C 180,E1 -9789.032,E2 -9789.032} C_VEL
LIN {X 0,Y 426.621,Z 337.61,A -85,B 0,C 180,E1 -9790.962,E2 -9790.962} C_VEL
LIN {X 0,Y 429.73,Z 358.15,A -85,B 0,C 180,E1 -9791.543,E2 -9791.543} C_VEL
LIN {X 0,Y 430.71,Z 368.012,A -85,B 0,C 180,E1 -9791.79,E2 -9791.79} C_VEL
LIN {X 0,Y 429.421,Z 448.753,A -85,B 0,C 180,E1 -9793.33,E2 -9793.33} C_VEL
LIN {X 0,Y 428.862,Z 462.011,A -85,B 0,C 180,E1 -9793.766,E2 -9793.766} C_VEL
LIN {X 0,Y 428.254,Z 474.257,A -85,B 0,C 180,E1 -9794.354,E2 -9794.354} C_VEL
LIN {X 0,Y 427.539,Z 486.14,A -85,B 0,C 180,E1 -9795.12,E2 -9795.12} C_VEL
LIN {X 0,Y 426.767,Z 498.038,A -85,B 0,C 180,E1 -9796.103,E2 -9796.103} C_VEL
LIN {X 0,Y 426.134,Z 508.068,A -85,B 0,C 180,E1 -9797.138,E2 -9797.138} C_VEL
LIN {X 0,Y 425.56,Z 517.454,A -85,B 0,C 180,E1 -9798.331,E2 -9798.331} C_VEL
LIN {X 0,Y 424.935,Z 526.609,A -85,B 0,C 180,E1 -9799.761,E2 -9799.761} C_VEL
LIN {X 0,Y 424.595,Z 534.001,A -85,B 0,C 180,E1 -9801.195,E2 -9801.195} C_VEL
LIN {X 0,Y 424.359,Z 539.008,A -85,B 0,C 180,E1 -9802.389,E2 -9802.389} C_VEL
LIN {X 0,Y 424.242,Z 543.513,A -85,B 0,C 180,E1 -9803.703,E2 -9803.703} C_VEL
LIN {X 0,Y 424.217,Z 547.608,A -85,B 0,C 180,E1 -9805.25,E2 -9805.25} C_VEL
LIN {X 0,Y 424.138,Z 549.511,A -85,B 0,C 180,E1 -9806.202,E2 -9806.202} C_VEL
LIN {X 0,Y 424.227,Z 550.955,A -85,B 0,C 180,E1 -9807.153,E2 -9807.153} C_VEL
LIN {X 0,Y 424.197,Z 551.986,A -85,B 0,C 180,E1 -9808.103,E2 -9808.103} C_VEL
LIN {X 0,Y 424.178,Z 552.615,A -85,B 0,C 180,E1 -9809.052,E2 -9809.052} C_VEL
LIN {X 0,Y 424.21,Z 552.8,A -85,B 0,C 180,E1 -9810.002,E2 -9810.002} C_VEL
LIN {X 0,Y 424.192,Z 552.558,A -85,B 0,C 180,E1 -9810.951,E2 -9810.951} C_VEL
LIN {X 0,Y 424.197,Z 551.916,A -85,B 0,C 180,E1 -9811.9,E2 -9811.9} C_VEL
LIN {X 0,Y 424.246,Z 550.87,A -85,B 0,C 180,E1 -9812.85,E2 -9812.85} C_VEL
LIN {X 0,Y 424.142,Z 549.343,A -85,B 0,C 180,E1 -9813.801,E2 -9813.801} C_VEL
LIN {X 0,Y 424.231,Z 546.243,A -85,B 0,C 180,E1 -9815.229,E2 -9815.229} C_VEL
LIN {X 0,Y 424.301,Z 542.039,A -85,B 0,C 180,E1 -9816.659,E2 -9816.659} C_VEL
LIN {X 0,Y 424.502,Z 535.595,A -85,B 0,C 180,E1 -9818.33,E2 -9818.33} C_VEL
LIN {X 0,Y 424.807,Z 528.558,A -85,B 0,C 180,E1 -9819.764,E2 -9819.764} C_VEL
LIN {X 0,Y 425.31,Z 519.724,A -85,B 0,C 180,E1 -9821.196,E2 -9821.196} C_VEL
LIN {X 0,Y 425.867,Z 509.671,A -85,B 0,C 180,E1 -9822.51,E2 -9822.51} C_VEL
LIN {X 0,Y 426.426,Z 499.716,A -85,B 0,C 180,E1 -9823.559,E2 -9823.559} C_VEL
LIN {X 0,Y 427.126,Z 488.129,A -85,B 0,C 180,E1 -9824.532,E2 -9824.532} C_VEL
LIN {X 0,Y 427.697,Z 477.437,A -85,B 0,C 180,E1 -9825.243,E2 -9825.243} C_VEL
LIN {X 0,Y 428.307,Z 464.608,A -85,B 0,C 180,E1 -9825.892,E2 -9825.892} C_VEL
LIN {X 0,Y 428.808,Z 451.867,A -85,B 0,C 180,E1 -9826.331,E2 -9826.331} C_VEL
LIN {X 0,Y 429.101,Z 432.938,A -85,B 0,C 180,E1 -9826.717,E2 -9826.717} C_VEL
LIN {X 0,Y 429.922,Z 365.317,A -85,B 0,C 180,E1 -9827.957,E2 -9827.957} C_VEL
LIN {X 0,Y 426.446,Z 340.108,A -85,B 0,C 180,E1 -9828.59,E2 -9828.59} C_VEL
LIN {X 0,Y 427.488,Z 321.434,A -85,B 0,C 180,E1 -9831.963,E2 -9831.963} C_VEL
LIN {X 0,Y 428.548,Z 303.55,A -85,B 0,C 180,E1 -9835.238,E2 -9835.238} C_VEL
LIN {X 0,Y 425.341,Z 287.504,A -85,B 0,C 180,E1 -9838.478,E2 -9838.478} C_VEL
LIN {X 0,Y 425.257,Z 287.512,A -85,B 0,C 180,E1 -9841.926,E2 -9841.926} C_VEL
LIN {X 0,Y 425.287,Z 287.506,A -85,B 0,C 180,E1 -9845.335,E2 -9845.335} C_VEL
LIN {X 0,Y 425.268,Z 287.513,A -85,B 0,C 180,E1 -9848.899,E2 -9848.899} C_VEL
LIN {X 0,Y 425.246,Z 287.517,A -85,B 0,C 180,E1 -9852.653,E2 -9852.653} C_VEL
LIN {X 0,Y 425.27,Z 287.51,A -85,B 0,C 180,E1 -9855.281,E2 -9855.281} C_VEL
LIN {X 0,Y 425.232,Z 287.517,A -85,B 0,C 180,E1 -9858.616,E2 -9858.616} C_VEL
LIN {X 0,Y 425.26,Z 287.513,A -85,B 0,C 180,E1 -9861.097,E2 -9861.097} C_VEL
LIN {X 0,Y 425.274,Z 287.512,A -85,B 0,C 180,E1 -9864.661,E2 -9864.661} C_VEL
LIN {X 0,Y 425.237,Z 287.513,A -85,B 0,C 180,E1 -9868.07,E2 -9868.07} C_VEL
LIN {X 0,Y 425.306,Z 287.506,A -85,B 0,C 180,E1 -9871.366,E2 -9871.366} C_VEL
LIN {X 0,Y 425.243,Z 287.514,A -85,B 0,C 180,E1 -9874.551,E2 -9874.551} C_VEL
LIN {X 0,Y 425.261,Z 287.511,A -85,B 0,C 180,E1 -9877.659,E2 -9877.659} C_VEL
LIN {X 0,Y 425.332,Z 287.504,A -85,B 0,C 180,E1 -9880.702,E2 -9880.702} C_VEL
LIN {X 0,Y 425.357,Z 287.499,A -85,B 0,C 180,E1 -9883.687,E2 -9883.687} C_VEL
LIN {X 0,Y 425.384,Z 287.496,A -85,B 0,C 180,E1 -9887.597,E2 -9887.597} C_VEL
LIN {X 0,Y 425.411,Z 287.493,A -85,B 0,C 180,E1 -9891.449,E2 -9891.449} C_VEL
LIN {X 0,Y 425.514,Z 287.48,A -85,B 0,C 180,E1 -9894.312,E2 -9894.312} C_VEL
LIN {X 0,Y 425.538,Z 287.478,A -85,B 0,C 180,E1 -9898.107,E2 -9898.107} C_VEL
LIN {X 0,Y 425.666,Z 287.461,A -85,B 0,C 180,E1 -9900,E2 -9900} C_VEL
LIN {X 0,Y 425.51,Z 287.482,A -85,B 0,C 180,E1 -9902.84,E2 -9902.84} C_VEL
LIN {X 0,Y 425.491,Z 287.483,A -85,B 0,C 180,E1 -9906.639,E2 -9906.639} C_VEL
LIN {X 0,Y 425.372,Z 287.499,A -85,B 0,C 180,E1 -9909.51,E2 -9909.51} C_VEL
LIN {X 0,Y 425.373,Z 287.499,A -85,B 0,C 180,E1 -9912.91,E2 -9912.91} C_VEL
LIN {X 0,Y 425.33,Z 287.503,A -85,B 0,C 180,E1 -9916.605,E2 -9916.605} C_VEL
LIN {X 0,Y 425.298,Z 287.508,A -85,B 0,C 180,E1 -9919.636,E2 -9919.636} C_VEL
LIN {X 0,Y 425.277,Z 287.512,A -85,B 0,C 180,E1 -9923.366,E2 -9923.366} C_VEL
LIN {X 0,Y 425.32,Z 287.505,A -85,B 0,C 180,E1 -9926.845,E2 -9926.845} C_VEL
LIN {X 0,Y 425.292,Z 287.508,A -85,B 0,C 180,E1 -9929.719,E2 -9929.719} C_VEL
LIN {X 0,Y 425.258,Z 287.513,A -85,B 0,C 180,E1 -9933.049,E2 -9933.049} C_VEL
LIN {X 0,Y 425.262,Z 287.512,A -85,B 0,C 180,E1 -9935.93,E2 -9935.93} C_VEL
LIN {X 0,Y 425.291,Z 287.508,A -85,B 0,C 180,E1 -9939.047,E2 -9939.047} C_VEL
LIN {X 0,Y 425.296,Z 287.508,A -85,B 0,C 180,E1 -9941.963,E2 -9941.963} C_VEL
LIN {X 0,Y 425.286,Z 287.509,A -85,B 0,C 180,E1 -9945.282,E2 -9945.282} C_VEL
LIN {X 0,Y 425.295,Z 287.51,A -85,B 0,C 180,E1 -9948.627,E2 -9948.627} C_VEL
LIN {X 0,Y 425.311,Z 287.506,A -85,B 0,C 180,E1 -9951.105,E2 -9951.105} C_VEL
LIN {X 0,Y 425.289,Z 287.511,A -85,B 0,C 180,E1 -9954.665,E2 -9954.665} C_VEL
LIN {X 0,Y 425.254,Z 287.513,A -85,B 0,C 180,E1 -9958.074,E2 -9958.074} C_VEL
LIN {X 0,Y 425.323,Z 287.504,A -85,B 0,C 180,E1 -9961.369,E2 -9961.369} C_VEL
LIN {X 0,Y 425.289,Z 287.511,A -85,B 0,C 180,E1 -9964.555,E2 -9964.555} C_VEL
LIN {X 0,Y 425.283,Z 287.51,A -85,B 0,C 180,E1 -9967.662,E2 -9967.662} C_VEL
LIN {X 0,Y 425.358,Z 287.503,A -85,B 0,C 180,E1 -9970.704,E2 -9970.704} C_VEL
LIN {X 0,Y 425.385,Z 287.497,A -85,B 0,C 180,E1 -9973.688,E2 -9973.688} C_VEL
LIN {X 0,Y 425.409,Z 287.493,A -85,B 0,C 180,E1 -9977.598,E2 -9977.598} C_VEL
LIN {X 0,Y 425.44,Z 287.489,A -85,B 0,C 180,E1 -9981.449,E2 -9981.449} C_VEL
LIN {X 0,Y 425.552,Z 287.475,A -85,B 0,C 180,E1 -9984.312,E2 -9984.312} C_VEL
LIN {X 0,Y 425.572,Z 287.472,A -85,B 0,C 180,E1 -9988.106,E2 -9988.106} C_VEL
LIN {X 0,Y 425.701,Z 287.456,A -85,B 0,C 180,E1 -9989.998,E2 -9989.998} C_VEL
LIN {X 0,Y 425.554,Z 287.479,A -85,B 0,C 180,E1 -9992.838,E2 -9992.838} C_VEL
LIN {X 0,Y 425.518,Z 287.481,A -85,B 0,C 180,E1 -9996.637,E2 -9996.637} C_VEL
LIN {X 0,Y 425.398,Z 287.493,A -85,B 0,C 180,E1 -9999.178,E2 -9999.178} C_VEL
LIN {X 0,Y 424.728,Z 287.578,A -85,B 0,C 180,E1 -9999.968,E2 -9999.968} C_VEL
LIN {X 0,Y 421.88,Z 287.938,A -85,B 0,C 180,E1 -10001.252,E2 -10001.252} C_VEL
LIN {X 0,Y 419.464,Z 288.239,A -85,B 0,C 180,E1 -10002.288,E2 -10002.288} C_VEL
LIN {X 0,Y 418.416,Z 288.367,A -85,B 0,C 180,E1 -10003.089,E2 -10003.089} C_VEL
LIN {X 0,Y 418.324,Z 288.376,A -85,B 0,C 180,E1 -10003.36,E2 -10003.36} C_VEL
LIN {X 0,Y 418.303,Z 288.38,A -85,B 0,C 180,E1 -10006.733,E2 -10006.733} C_VEL
LIN {X 0,Y 418.291,Z 288.378,A -85,B 0,C 180,E1 -10009.799,E2 -10009.799} C_VEL
LIN {X 0,Y 418.23,Z 288.388,A -85,B 0,C 180,E1 -10012.732,E2 -10012.732} C_VEL
LIN {X 0,Y 418.255,Z 288.382,A -85,B 0,C 180,E1 -10015.901,E2 -10015.901} C_VEL
LIN {X 0,Y 418.257,Z 288.388,A -85,B 0,C 180,E1 -10019.158,E2 -10019.158} C_VEL
LIN {X 0,Y 418.239,Z 288.387,A -85,B 0,C 180,E1 -10022.841,E2 -10022.841} C_VEL
LIN {X 0,Y 418.224,Z 288.385,A -85,B 0,C 180,E1 -10026.235,E2 -10026.235} C_VEL
LIN {X 0,Y 418.24,Z 288.389,A -85,B 0,C 180,E1 -10029.676,E2 -10029.676} C_VEL
LIN {X 0,Y 418.282,Z 288.466,A -85,B 0,C 180,E1 -10031.695,E2 -10031.695} C_VEL
LIN {X 0,Y 419.519,Z 294.867,A -85,B 0,C 180,E1 -10033.225,E2 -10033.225} C_VEL
LIN {X 0,Y 423.04,Z 310.559,A -85,B 0,C 180,E1 -10033.685,E2 -10033.685} C_VEL
LIN {X 0,Y 423.579,Z 313.281,A -85,B 0,C 180,E1 -10033.76,E2 -10033.76} C_VEL
LIN {X 0,Y 422.225,Z 402.973,A -85,B 0,C 180,E1 -10035.458,E2 -10035.458} C_VEL
LIN {X 0,Y 421.935,Z 416.303,A -85,B 0,C 180,E1 -10035.908,E2 -10035.908} C_VEL
LIN {X 0,Y 421.421,Z 429.058,A -85,B 0,C 180,E1 -10036.535,E2 -10036.535} C_VEL
LIN {X 0,Y 420.868,Z 441.305,A -85,B 0,C 180,E1 -10037.354,E2 -10037.354} C_VEL
LIN {X 0,Y 420.274,Z 452.248,A -85,B 0,C 180,E1 -10038.287,E2 -10038.287} C_VEL
LIN {X 0,Y 419.659,Z 462.558,A -85,B 0,C 180,E1 -10039.381,E2 -10039.381} C_VEL
LIN {X 0,Y 419.006,Z 472.784,A -85,B 0,C 180,E1 -10040.738,E2 -10040.738} C_VEL
LIN {X 0,Y 418.476,Z 481.152,A -85,B 0,C 180,E1 -10042.113,E2 -10042.113} C_VEL
LIN {X 0,Y 418.021,Z 488.402,A -85,B 0,C 180,E1 -10043.604,E2 -10043.604} C_VEL
LIN {X 0,Y 417.701,Z 494.2,A -85,B 0,C 180,E1 -10045.106,E2 -10045.106} C_VEL
LIN {X 0,Y 417.441,Z 499.288,A -85,B 0,C 180,E1 -10046.828,E2 -10046.828} C_VEL
LIN {X 0,Y 417.164,Z 502.794,A -85,B 0,C 180,E1 -10048.517,E2 -10048.517} C_VEL
LIN {X 0,Y 417.063,Z 504.37,A -85,B 0,C 180,E1 -10049.634,E2 -10049.634} C_VEL
LIN {X 0,Y 417.018,Z 505.654,A -85,B 0,C 180,E1 -10051.192,E2 -10051.192} C_VEL
LIN {X 0,Y 417.033,Z 505.851,A -85,B 0,C 180,E1 -10052.935,E2 -10052.935} C_VEL
LIN {X 0,Y 417.073,Z 505.269,A -85,B 0,C 180,E1 -10054.017,E2 -10054.017} C_VEL
LIN {X 0,Y 417.23,Z 503.76,A -85,B 0,C 180,E1 -10055.434,E2 -10055.434} C_VEL
LIN {X 0,Y 417.5,Z 500.535,A -85,B 0,C 180,E1 -10057.222,E2 -10057.222} C_VEL
LIN {X 0,Y 417.731,Z 496.426,A -85,B 0,C 180,E1 -10058.795,E2 -10058.795} C_VEL
LIN {X 0,Y 418.154,Z 490.989,A -85,B 0,C 180,E1 -10060.358,E2 -10060.358} C_VEL
LIN {X 0,Y 418.673,Z 484.038,A -85,B 0,C 180,E1 -10061.908,E2 -10061.908} C_VEL
LIN {X 0,Y 419.355,Z 475.338,A -85,B 0,C 180,E1 -10063.447,E2 -10063.447} C_VEL
LIN {X 0,Y 420.012,Z 466.311,A -85,B 0,C 180,E1 -10064.72,E2 -10064.72} C_VEL
LIN {X 0,Y 420.826,Z 455.411,A -85,B 0,C 180,E1 -10065.955,E2 -10065.955} C_VEL
LIN {X 0,Y 421.443,Z 445.45,A -85,B 0,C 180,E1 -10066.868,E2 -10066.868} C_VEL
LIN {X 0,Y 422.103,Z 433.274,A -85,B 0,C 180,E1 -10067.744,E2 -10067.744} C_VEL
LIN {X 0,Y 422.635,Z 420.661,A -85,B 0,C 180,E1 -10068.429,E2 -10068.429} C_VEL
LIN {X 0,Y 423.023,Z 407.932,A -85,B 0,C 180,E1 -10068.915,E2 -10068.915} C_VEL
LIN {X 0,Y 423.351,Z 391.428,A -85,B 0,C 180,E1 -10069.287,E2 -10069.287} C_VEL
LIN {X 0,Y 424.688,Z 313.203,A -85,B 0,C 180,E1 -10070.813,E2 -10070.813} C_VEL
LIN {X 0,Y 421.903,Z 300.333,A -85,B 0,C 180,E1 -10071.239,E2 -10071.239} C_VEL
LIN {X 0,Y 419.93,Z 295.096,A -85,B 0,C 180,E1 -10071.489,E2 -10071.489} C_VEL
LIN {X 0,Y 418.402,Z 288.37,A -85,B 0,C 180,E1 -10072.813,E2 -10072.813} C_VEL
LIN {X 0,Y 418.454,Z 288.365,A -85,B 0,C 180,E1 -10074.217,E2 -10074.217} C_VEL
LIN {X 0,Y 418.49,Z 288.358,A -85,B 0,C 180,E1 -10078.076,E2 -10078.076} C_VEL
LIN {X 0,Y 418.616,Z 288.339,A -85,B 0,C 180,E1 -10080,E2 -10080} C_VEL
LIN {X 0,Y 418.462,Z 288.361,A -85,B 0,C 180,E1 -10082.889,E2 -10082.889} C_VEL
LIN {X 0,Y 418.436,Z 288.363,A -85,B 0,C 180,E1 -10086.752,E2 -10086.752} C_VEL
LIN {X 0,Y 418.293,Z 288.379,A -85,B 0,C 180,E1 -10089.673,E2 -10089.673} C_VEL
LIN {X 0,Y 418.305,Z 288.379,A -85,B 0,C 180,E1 -10093.008,E2 -10093.008} C_VEL
LIN {X 0,Y 418.263,Z 288.385,A -85,B 0,C 180,E1 -10096.737,E2 -10096.737} C_VEL
LIN {X 0,Y 418.221,Z 288.384,A -85,B 0,C 180,E1 -10099.792,E2 -10099.792} C_VEL
LIN {X 0,Y 418.192,Z 288.392,A -85,B 0,C 180,E1 -10102.739,E2 -10102.739} C_VEL
LIN {X 0,Y 418.226,Z 288.383,A -85,B 0,C 180,E1 -10105.907,E2 -10105.907} C_VEL
LIN {X 0,Y 418.224,Z 288.388,A -85,B 0,C 180,E1 -10109.166,E2 -10109.166} C_VEL
LIN {X 0,Y 418.218,Z 288.389,A -85,B 0,C 180,E1 -10112.847,E2 -10112.847} C_VEL
LIN {X 0,Y 418.212,Z 288.388,A -85,B 0,C 180,E1 -10116.242,E2 -10116.242} C_VEL
LIN {X 0,Y 418.232,Z 288.386,A -85,B 0,C 180,E1 -10119.685,E2 -10119.685} C_VEL
LIN {X 0,Y 418.215,Z 288.385,A -85,B 0,C 180,E1 -10122.328,E2 -10122.328} C_VEL
LIN {X 0,Y 418.208,Z 288.391,A -85,B 0,C 180,E1 -10125.113,E2 -10125.113} C_VEL
LIN {X 0,Y 418.214,Z 288.391,A -85,B 0,C 180,E1 -10127.771,E2 -10127.771} C_VEL
LIN {X 0,Y 418.219,Z 288.388,A -85,B 0,C 180,E1 -10130.626,E2 -10130.626} C_VEL
LIN {X 0,Y 418.223,Z 288.392,A -85,B 0,C 180,E1 -10133.98,E2 -10133.98} C_VEL
LIN {X 0,Y 418.241,Z 288.396,A -85,B 0,C 180,E1 -10137.16,E2 -10137.16} C_VEL
LIN {X 0,Y 418.248,Z 288.392,A -85,B 0,C 180,E1 -10140.842,E2 -10140.842} C_VEL
LIN {X 0,Y 418.273,Z 288.413,A -85,B 0,C 180,E1 -10141.804,E2 -10141.804} C_VEL
